// TwinCAT 3 PLC project SPS_Demonstrator
// ProgramVersion: 3.1.4026.19
// libraries:
//   Tc2_Standard, * (Beckhoff Automation GmbH)
//   Tc2_System, * (Beckhoff Automation GmbH)
//   Tc3_EventLogger, * (Beckhoff Automation GmbH)
//   Tc3_Module, * (Beckhoff Automation GmbH)
// project tree:
//   GVLs/ GVL.TcGVL, GVL_HRL.TcGVL, GVL_MBS.TcGVL, GVL_SST.TcGVL, GVL_VSG.TcGVL
//   / PlcTask.TcTTO
//   POUs/AtomicSkills/ Auto_ColorDetection.TcPOU, AxisControl_MultipleInputSensors.TcPOU, AxisControl_Encoder.TcPOU, CompressorControl.TcPOU, SecuringWorkpiece.TcPOU, StampingProcess.TcPOU, HardeningProcess.TcPOU, CuttingProcess.TcPOU
//   POUs/ControlOfOutputs/ HRL_ControlOfOutputs.TcPOU, MBS_ControlOfOutputs.TcPOU, SST_ControlOfOutputs.TcPOU, VSG_ControlOfOutputs.TcPOU
//   POUs/ HRL_SkillSet.TcPOU
//   POUs/MethodenBeispiele/ FB_MyOpcUaMethod.TcPOU, JobMethode_Schablone.TcPOU, HRL_NMethod_Auslagern.TcPOU, JobMethode.TcPOU
//   POUs/Moduls/HRL_Skills/ HRL_RGB_AS_VerticalMoveEncoder.TcPOU, HRL_RGB_AS_HorizontalMoveSensors.TcPOU, HRL_CB_AS_HorizontalMove.TcPOU, HRL_RGB_AS_HorizontalMoveEncoder.TcPOU, HRL_RGB_InitalStateDrive.TcPOU
//   POUs/Moduls/MBS_Skills/ MBS_MR01_AS_HardeningProcess.TcPOU, MBS_MR01_AS_SecuringProcess.TcPOU, MBS_VSG_AS_VerticalMove.TcPOU, MBS_MR01_AS_HorizontalMove.TcPOU, MBS_DmPD_AS_RotationMove.TcPOU, MBS_VSG_AS_HorizontalMove.TcPOU, MBS_CB_AS_HorizontalMove.TcPOU, MBS_DmPD_AS_HorizontalMove.TcPOU, MBS_MR02_AS_CuttingProcess.TcPOU
//   POUs/Moduls/SST_Skills/ SST_PD_AS_HorizontalMove.TcPOU, SST_CB_AS_HorizontalMove.TcPOU, SST_CS_AS_ColorDetection.TcPOU
//   POUs/Moduls/VSG_Skills/ VSG_AS_HorizontalMoveEncoder.TcPOU, VSG_AS_VerticalMoveEncoder.TcPOU, VSG_AS_RotationMoveEncoder.TcPOU, VSG_AS_CompressorControl.TcPOU
//   POUs/OperatingModes/ HRL_OperatingModes.TcPOU, MBS_OperatingModes.TcPOU, SST_OperatingModes.TcPOU, SVG_OperatingModes.TcPOU
// real-time tasks:
//   TASK PlcTask: cycle T#10ms, priority 20, ADS port 350
// I/O:
//   DEVICE Gerät 1 (EtherCAT), AmsNetId 5.152.132.139.2.1
//     Klemme 1 (EK1200) [EK1200-5000 EtherCAT Netzteil (2A E-Bus)]
//       Klemme 2 (EL1512) [EL1512 2K. +/- Zaehler 24V, 1kHz]
//       Klemme 3 (EL1512) [EL1512 2K. +/- Zaehler 24V, 1kHz]
//       Klemme 4 (EL1512) [EL1512 2K. +/- Zaehler 24V, 1kHz]
//       Klemme 5 (EL1512) [EL1512 2K. +/- Zaehler 24V, 1kHz]
//       Klemme 6 (EL1512) [EL1512 2K. +/- Zaehler 24V, 1kHz]
//       Klemme 7 (EL1409) [EL1409 16K. Dig. Eingang 24V, 3ms]
//       Klemme 8 (EL1409) [EL1409 16K. Dig. Eingang 24V, 3ms]
//       Klemme 9 (EL2409) [EL2409 16K. Dig. Ausgang 24V, 0.5A]
//       Klemme 10 (EL2409) [EL2409 16K. Dig. Ausgang 24V, 0.5A]
//       Klemme 11 (EL2008) [EL2008 8K. Dig. Ausgang 24V, 0.5A]
//       Klemme 12 (EL3072) [EL3072 2K. Ana. Eingang  +/-10V, +/-20mA]
//       Klemme 13 (EL9011) [EL9011 Endklemme]
// variable links:
//   SPS_Demonstrator/SPS_Demonstrator Instance <-> Device 1 (EtherCAT)/Term 1 (EK1200)/Term 10 (EL2409)
//     PlcTask Outputs/GVL_MBS.MBS_Kompressor <-> Channel 2/Output
//     PlcTask Outputs/GVL_MBS.MBS_Leuchte_Ofen <-> Channel 1/Output
//     PlcTask Outputs/GVL_MBS.MBS_MV_Ofentuer <-> Channel 5/Output
//     PlcTask Outputs/GVL_MBS.MBS_MV_Schieber <-> Channel 6/Output
//     PlcTask Outputs/GVL_MBS.MBS_MV_Vakuum <-> Channel 3/Output
//     PlcTask Outputs/GVL_MBS.MBS_MV_senken <-> Channel 4/Output
//     PlcTask Outputs/GVL_SST.SST_Kompressor <-> Channel 16/Output
//     PlcTask Outputs/GVL_SST.SST_MOT_Foerderband <-> Channel 15/Output
//     PlcTask Outputs/GVL_VSG.VSG_Kompressor <-> Channel 13/Output
//     PlcTask Outputs/GVL_VSG.VSG_MOT_drehen_CCW <-> Channel 12/Output
//     PlcTask Outputs/GVL_VSG.VSG_MOT_drehen_CW <-> Channel 11/Output
//     PlcTask Outputs/GVL_VSG.VSG_MOT_horizontal_rueckwaerts <-> Channel 9/Output
//     PlcTask Outputs/GVL_VSG.VSG_MOT_horizontal_vorwaerts <-> Channel 10/Output
//     PlcTask Outputs/GVL_VSG.VSG_MOT_vertikal_hoch <-> Channel 7/Output
//     PlcTask Outputs/GVL_VSG.VSG_MOT_vertikal_runter <-> Channel 8/Output
//     PlcTask Outputs/GVL_VSG.VSG_MV_Vakuum <-> Channel 14/Output
//   SPS_Demonstrator/SPS_Demonstrator Instance <-> Device 1 (EtherCAT)/Term 1 (EK1200)/Term 11 (EL2008)
//     PlcTask Outputs/GVL_SST.SST_MV_blau <-> Channel 3/Output
//     PlcTask Outputs/GVL_SST.SST_MV_rot <-> Channel 2/Output
//     PlcTask Outputs/GVL_SST.SST_MV_weiss <-> Channel 1/Output
//   SPS_Demonstrator/SPS_Demonstrator Instance <-> Device 1 (EtherCAT)/Term 1 (EK1200)/Term 12 (EL3072)
//     PlcTask Inputs/GVL_SST.SST_Farbsensor <-> AI Standard Channel 1/Value
//   SPS_Demonstrator/SPS_Demonstrator Instance <-> Device 1 (EtherCAT)/Term 1 (EK1200)/Term 2 (EL1512)
//     PlcTask Inputs/GVL_HRL.HRL_Enc_horizontal_I1 <-> CNT Inputs Channel 1/Counter value
//     PlcTask Inputs/GVL_HRL.HRL_Enc_horizontal_I2 <-> CNT Inputs Channel 2/Counter value
//     PlcTask Outputs/GVL_HRL.HRL_K1_1_Zaehler_Zuruecksetzen <-> CNT Outputs Channel 1/Control/Set counter
//   SPS_Demonstrator/SPS_Demonstrator Instance <-> Device 1 (EtherCAT)/Term 1 (EK1200)/Term 3 (EL1512)
//     PlcTask Inputs/GVL_HRL.HRL_Enc_vertikal_I1 <-> CNT Inputs Channel 1/Counter value
//     PlcTask Inputs/GVL_HRL.HRL_Enc_vertikal_I2 <-> CNT Inputs Channel 2/Counter value
//     PlcTask Outputs/GVL_HRL.HRL_K1_2_Zaehler_Zuruecksetzen <-> CNT Outputs Channel 1/Control/Set counter
//   SPS_Demonstrator/SPS_Demonstrator Instance <-> Device 1 (EtherCAT)/Term 1 (EK1200)/Term 4 (EL1512)
//     PlcTask Inputs/GVL_VSG.VSG_Enc_vertikal_I1 <-> CNT Inputs Channel 1/Counter value
//     PlcTask Inputs/GVL_VSG.VSG_Enc_vertikal_I2 <-> CNT Inputs Channel 2/Counter value
//     PlcTask Outputs/GVL_VSG.VSG_K1_3_Zaehler_Zuruecksetzen <-> CNT Outputs Channel 1/Control/Set counter
//   SPS_Demonstrator/SPS_Demonstrator Instance <-> Device 1 (EtherCAT)/Term 1 (EK1200)/Term 5 (EL1512)
//     PlcTask Inputs/GVL_VSG.VSG_Enc_horizontal_I1 <-> CNT Inputs Channel 1/Counter value
//     PlcTask Inputs/GVL_VSG.VSG_Enc_horizontal_I2 <-> CNT Inputs Channel 2/Counter value
//     PlcTask Outputs/GVL_VSG.VSG_K1_4_Zaehler_Zuruecksetzen <-> CNT Outputs Channel 1/Set counter
//   SPS_Demonstrator/SPS_Demonstrator Instance <-> Device 1 (EtherCAT)/Term 1 (EK1200)/Term 6 (EL1512)
//     PlcTask Inputs/GVL_VSG.VSG_Enc_drehen_I1 <-> CNT Inputs Channel 1/Counter value
//     PlcTask Inputs/GVL_VSG.VSG_Enc_drehen_I2 <-> CNT Inputs Channel 2/Counter value
//     PlcTask Outputs/GVL_VSG.VSG_K1_5_Zaehler_Zuruecksetzen <-> CNT Outputs Channel 1/Control/Set counter
//   SPS_Demonstrator/SPS_Demonstrator Instance <-> Device 1 (EtherCAT)/Term 1 (EK1200)/Term 7 (EL1409)
//     PlcTask Inputs/GVL_HRL.HRL_LS_aussen <-> DIP Inputs/Input Channel 3
//     PlcTask Inputs/GVL_HRL.HRL_LS_innen <-> DIP Inputs/Input Channel 2
//     PlcTask Inputs/GVL_HRL.HRL_Ref_Taster_Ausleger_hinten <-> DIP Inputs/Input Channel 8
//     PlcTask Inputs/GVL_HRL.HRL_Ref_Taster_Ausleger_vorne <-> DIP Inputs/Input Channel 7
//     PlcTask Inputs/GVL_HRL.HRL_Ref_Taster_horizontal <-> DIP Inputs/Input Channel 1
//     PlcTask Inputs/GVL_HRL.HRL_Ref_Taster_vertikal <-> DIP Inputs/Input Channel 4
//     PlcTask Inputs/GVL_HRL.HRL_Spursensor_1_unten <-> DIP Inputs/Input Channel 5
//     PlcTask Inputs/GVL_HRL.HRL_Spursensor_2_oben <-> DIP Inputs/Input Channel 6
//     PlcTask Inputs/GVL_MBS.MBS_LS_Ende_Foerderband <-> DIP Inputs/Input Channel 11
//     PlcTask Inputs/GVL_MBS.MBS_Ref_Taster_DK_Pos_Foerderband <-> DIP Inputs/Input Channel 10
//     PlcTask Inputs/GVL_MBS.MBS_Ref_Taster_DK_Pos_Saege <-> DIP Inputs/Input Channel 12
//     PlcTask Inputs/GVL_MBS.MBS_Ref_Taster_DK_Pos_Sauger <-> DIP Inputs/Input Channel 9
//     PlcTask Inputs/GVL_MBS.MBS_Ref_Taster_Ofenschieber_aussen <-> DIP Inputs/Input Channel 15
//     PlcTask Inputs/GVL_MBS.MBS_Ref_Taster_Ofenschieber_innen <-> DIP Inputs/Input Channel 14
//     PlcTask Inputs/GVL_MBS.MBS_Ref_Taster_Sauger_Pos_DK <-> DIP Inputs/Input Channel 13
//     PlcTask Inputs/GVL_MBS.MBS_Ref_Taster_Sauger_Pos_Ofen <-> DIP Inputs/Input Channel 16
//   SPS_Demonstrator/SPS_Demonstrator Instance <-> Device 1 (EtherCAT)/Term 1 (EK1200)/Term 8 (EL1409)
//     PlcTask Inputs/GVL.diNotAus_Kanal_A <-> DIP Inputs/Input Channel 11
//     PlcTask Inputs/GVL.diNotAus_Kanal_B <-> DIP Inputs/Input Channel 12
//     PlcTask Inputs/GVL_MBS.MBS_LS_Ofen <-> DIP Inputs/Input Channel 1
//     PlcTask Inputs/GVL_SST.SST_Impulstaster <-> DIP Inputs/Input Channel 5
//     PlcTask Inputs/GVL_SST.SST_LS_Eingang <-> DIP Inputs/Input Channel 6
//     PlcTask Inputs/GVL_SST.SST_LS_blau <-> DIP Inputs/Input Channel 10
//     PlcTask Inputs/GVL_SST.SST_LS_nach_Farbsensor <-> DIP Inputs/Input Channel 7
//     PlcTask Inputs/GVL_SST.SST_LS_rot <-> DIP Inputs/Input Channel 9
//     PlcTask Inputs/GVL_SST.SST_LS_weiss <-> DIP Inputs/Input Channel 8
//     PlcTask Inputs/GVL_VSG.VSG_Ref_Schalter_drehen <-> DIP Inputs/Input Channel 4
//     PlcTask Inputs/GVL_VSG.VSG_Ref_Schalter_horizontal <-> DIP Inputs/Input Channel 3
//     PlcTask Inputs/GVL_VSG.VSG_Ref_Schalter_vertikal <-> DIP Inputs/Input Channel 2
//   SPS_Demonstrator/SPS_Demonstrator Instance <-> Device 1 (EtherCAT)/Term 1 (EK1200)/Term 9 (EL2409)
//     PlcTask Outputs/GVL_HRL.HRL_MOT_Ausleger_rueckwaerts <-> Channel 8/Output
//     PlcTask Outputs/GVL_HRL.HRL_MOT_Ausleger_vorwaerts <-> Channel 7/Output
//     PlcTask Outputs/GVL_HRL.HRL_MOT_Foerderband_rueckwaerts <-> Channel 2/Output
//     PlcTask Outputs/GVL_HRL.HRL_MOT_Foerderband_vorwaerts <-> Channel 1/Output
//     PlcTask Outputs/GVL_HRL.HRL_MOT_horizontal_zum_Foerderband <-> Channel 4/Output
//     PlcTask Outputs/GVL_HRL.HRL_MOT_horizontal_zum_Regal <-> Channel 3/Output
//     PlcTask Outputs/GVL_HRL.HRL_MOT_vertikal_hoch <-> Channel 6/Output
//     PlcTask Outputs/GVL_HRL.HRL_MOT_vertikal_runter <-> Channel 5/Output
//     PlcTask Outputs/GVL_MBS.MBS_MOT_DK_CCW <-> Channel 10/Output
//     PlcTask Outputs/GVL_MBS.MBS_MOT_DK_CW <-> Channel 9/Output
//     PlcTask Outputs/GVL_MBS.MBS_MOT_Foerderband_vorwaerts <-> Channel 11/Output
//     PlcTask Outputs/GVL_MBS.MBS_MOT_Ofenschieber_ausfahren <-> Channel 14/Output
//     PlcTask Outputs/GVL_MBS.MBS_MOT_Ofenschieber_einfahren <-> Channel 13/Output
//     PlcTask Outputs/GVL_MBS.MBS_MOT_Saege <-> Channel 12/Output
//     PlcTask Outputs/GVL_MBS.MBS_MOT_Sauger_zum_DK <-> Channel 16/Output
//     PlcTask Outputs/GVL_MBS.MBS_MOT_Sauger_zum_Ofen <-> Channel 15/Output

CONFIGURATION SPS_Demonstrator
    RESOURCE PLC ON TwinCAT3
        TASK PlcTask(INTERVAL := T#10ms, PRIORITY := 20);
        PROGRAM InitalizingOM WITH PlcTask : InitalizingOM;
        PROGRAM HRL_SkillSet WITH PlcTask : HRL_SkillSet;
    END_RESOURCE
END_CONFIGURATION

// ---- GVLs/GVL.TcGVL
{attribute 'qualified_only'}
VAR_GLOBAL
	// xDI%139.2_S1_2
	diNotAus_Kanal_A AT %I*: BOOL;
	// xDI%139.3_S1_2
	diNotAus_Kanal_B AT %I*: BOOL;
END_VAR

// ---- GVLs/GVL_HRL.TcGVL
{attribute 'qualified_only'}
VAR_GLOBAL
	// udiDI%41.0_A2_5
	HRL_Enc_horizontal_I1 AT %I*: UDINT;
	// udiDI%47.0_A2_5
	HRL_Enc_horizontal_I2 AT %I*: UDINT;
	// udiDI%53.0_A2_5
	HRL_Enc_vertikal_I1 AT %I*: UDINT;
	// udiDI%59.0_A2_5
	HRL_Enc_vertikal_I2 AT %I*: UDINT;
	// xDI%136.0_A2_2
	HRL_Ref_Taster_horizontal AT %I*: BOOL;
	// xDI%136.1_A2_1
	HRL_LS_innen AT %I*: BOOL;
	// xDI%136.2_A2_1
	HRL_LS_aussen AT %I*: BOOL;
	// xDI%136.3_A2_2
	HRL_Ref_Taster_vertikal AT %I*: BOOL;
	// xDI%136.4_A2_3
	HRL_Spursensor_1_unten AT %I*: BOOL;
	// xDI%136.5_A2_3
	HRL_Spursensor_2_oben AT %I*: BOOL;
	// xDI%136.6_A2_2
	HRL_Ref_Taster_Ausleger_vorne AT %I*: BOOL;
	// xDI%136.7_A2_2
	HRL_Ref_Taster_Ausleger_hinten AT %I*: BOOL;
	// xDO%111.0_A2_2	
	HRL_MOT_Foerderband_vorwaerts AT %Q*: BOOL;
	// xDO%111.1_A2_2
	HRL_MOT_Foerderband_rueckwaerts AT %Q*: BOOL;
	// xDO%111.2_A2_4
	HRL_MOT_horizontal_zum_Regal AT %Q*: BOOL;
	// xDO%111.3_A2_4
	HRL_MOT_horizontal_zum_Foerderband AT %Q*: BOOL;
	// xDO%111.4_A2_4
	HRL_MOT_vertikal_runter AT %Q*: BOOL;
	// xDO%111.5_A2_4
	HRL_MOT_vertikal_hoch AT %Q*: BOOL;
	// xDO%111.6_A2_4
	HRL_MOT_Ausleger_vorwaerts AT %Q*: BOOL;
	// xDO%111.7_A2_4
	HRL_MOT_Ausleger_rueckwaerts AT %Q*: BOOL;
	HRL_K1_1_Zaehler_Zuruecksetzen AT %Q*: BOOL;
	HRL_K1_2_Zaehler_Zuruecksetzen AT %Q*: BOOL;
END_VAR

// ---- GVLs/GVL_MBS.TcGVL
{attribute 'qualified_only'}
VAR_GLOBAL
	// xDI%137.0_A3_2
	MBS_Ref_Taster_DK_Pos_Sauger AT %I*: BOOL;
	// xDI%137.1_A3_2
	MBS_Ref_Taster_DK_Pos_Foerderband AT %I*: BOOL;
	// xDI%137.2_A3_1
	MBS_LS_Ende_Foerderband AT %I*: BOOL;
	// xDI%137.3_A3_2
	MBS_Ref_Taster_DK_Pos_Saege AT %I*: BOOL;
	// xDI%137.4_A3_2
	MBS_Ref_Taster_Sauger_Pos_DK AT %I*: BOOL;
	// xDI%137.5_A3_2
	MBS_Ref_Taster_Ofenschieber_innen AT %I*: BOOL;
	// xDI%137.6_A3_2
	MBS_Ref_Taster_Ofenschieber_aussen AT %I*: BOOL;
	// xDI%137.7_A3_2
	MBS_Ref_Taster_Sauger_Pos_Ofen AT %I*: BOOL;
	// xDI%138.0_A3_1
	MBS_LS_Ofen AT %I*: BOOL;
	// xDO%112.0_A3_4
	MBS_MOT_DK_CW AT %Q*: BOOL;
	// xDO%112.1_A3_4
	MBS_MOT_DK_CCW AT %Q*: BOOL;
	// xDO%112.2_A3_2
	MBS_MOT_Foerderband_vorwaerts AT %Q*: BOOL;
	// xDO%112.3_A3_6
	MBS_MOT_Saege AT %Q*: BOOL;
	// xDO%112.4_A3_3
	MBS_MOT_Ofenschieber_einfahren AT %Q*: BOOL;
	// xDO%112.5_A3_3
	MBS_MOT_Ofenschieber_ausfahren AT %Q*: BOOL;
	// xDO%112.6_A3_5
	MBS_MOT_Sauger_zum_Ofen AT %Q*: BOOL;
	// xDO%112.7_A3_5
	MBS_MOT_Sauger_zum_DK AT %Q*: BOOL;
	// xDO%113.0_A3_7
	MBS_Leuchte_Ofen AT %Q*: BOOL;
	// xDO%113.1_A3_8
	MBS_Kompressor AT %Q*: BOOL;
	// xDO%113.2_A3_5
	MBS_MV_Vakuum AT %Q*: BOOL;
	// xDO%113.3_A3_5
	MBS_MV_senken AT %Q*: BOOL;
	// xDO%113.4_A3_5
	MBS_MV_Ofentuer AT %Q*: BOOL;
	// xDO%113.5_A3_5
	MBS_MV_Schieber AT %Q*: BOOL;
END_VAR

// ---- GVLs/GVL_SST.TcGVL
{attribute 'qualified_only'}
VAR_GLOBAL
	// xDO%115.0_A5_5
	SST_MV_weiss AT %Q*: BOOL;
	// xDO%115.1_A5_5
	SST_MV_rot AT %Q*: BOOL;
	// xDO%115.2_A5_5
	SST_MV_blau AT %Q*: BOOL;
	// iAI%130.0_A5_4
	SST_Farbsensor AT %I*: INT;
	// xDI%138.4_A5_1
	SST_Impulstaster AT %I*: BOOL;
	// xDI%138.5_A5_1
	SST_LS_Eingang AT %I*: BOOL;
	// xDI%138.6_A5_1
	SST_LS_nach_Farbsensor AT %I*: BOOL;
	// xDI%138.7_A5_1
	SST_LS_weiss AT %I*: BOOL;
	// xDI%139.0_A5_1
	SST_LS_rot AT %I*: BOOL;
	// xDI%139.1_A5_1
	SST_LS_blau AT %I*: BOOL;
	// xDO%114.6_A5_2
	SST_MOT_Foerderband AT %Q*: BOOL;
	// xDO%114.7_A5_8
	SST_Kompressor AT %Q*: BOOL;
END_VAR

// ---- GVLs/GVL_VSG.TcGVL
{attribute 'qualified_only'}
VAR_GLOBAL
	// udiDI%65.0_A4_5
	VSG_Enc_vertikal_I1 AT %I*: UDINT;
	// udiDI%71.0_A4_5
	VSG_Enc_vertikal_I2 AT %I*: UDINT;
	// udiDI%77.0_A4_5
	VSG_Enc_horizontal_I1 AT %I*: UDINT;
	// udiDI%83.0_A4_5
	VSG_Enc_horizontal_I2 AT %I*: UDINT;
	// udiDI%89.0_A4_5
	VSG_Enc_drehen_I1 AT %I*: UDINT;
	// udiDI%95.0_A4_5
	VSG_Enc_drehen_I2 AT %I*: UDINT;
	// xDI%138.1_A4_2
	VSG_Ref_Schalter_vertikal AT %I*: BOOL;
	// xDI%138.2_A4_2
	VSG_Ref_Schalter_horizontal AT %I*: BOOL;
	// xDI%138.3_A4_2
	VSG_Ref_Schalter_drehen AT %I*: BOOL;
	// xDO%113.6_A4_4
	VSG_MOT_vertikal_hoch AT %Q*: BOOL;
	// xDO%113.7_A4_4
	VSG_MOT_vertikal_runter AT %Q*: BOOL;
	// xDO%114.0_A4_4
	VSG_MOT_horizontal_rueckwaerts AT %Q*: BOOL;
	// xDO%114.1_A4_4
	VSG_MOT_horizontal_vorwaerts AT %Q*: BOOL;
	// xDO%114.2_A4_4
	VSG_MOT_drehen_CW AT %Q*: BOOL;
	// xDO%114.3_A4_4
	VSG_MOT_drehen_CCW AT %Q*: BOOL;
	// xDO%114.4_A4_8
	VSG_Kompressor AT %Q*: BOOL;
	// xDO%114.5_A4_5
	VSG_MV_Vakuum AT %Q*: BOOL;
	VSG_K1_4_Zaehler_Zuruecksetzen AT %Q*: BOOL;
	VSG_K1_5_Zaehler_Zuruecksetzen AT %Q*: BOOL;
	VSG_K1_3_Zaehler_Zuruecksetzen AT %Q*: BOOL;
END_VAR

// ---- POUs/HRL_SkillSet.TcPOU
PROGRAM HRL_SkillSet
VAR
//Hochregallager Skillset	
	
	//HRL Conveyorbelt Skills
	{attribute 'OPC.UA.DA':= '1'}
	HRL_Skill_CB_MoveForwards: HRL_CB_AS_HorizontalMove; //Movement to Store-Out some goods on the Conveyorbelt
	{attribute 'OPC.UA.DA':= '1'}
	HRL_Skill_CB_MoveBackwards : HRL_CB_AS_HorizontalMove; //Movement to Store-In some goods on the Conveyorbelt
	
	//HRL RGB Skills
	{attribute 'OPC.UA.DA':= '1'}
	HRL_Skill_RGB_MoveBackwards : HRL_RGB_AS_HorizontalMoveSensors;	
	{attribute 'OPC.UA.DA':= '1'}
	HRL_Skill_RGB_MoveForwards : HRL_RGB_AS_HorizontalMoveSensors;	
	{attribute 'OPC.UA.DA':= '1'}
	HRL_Skill_RGB_MoveVerticalForwards : HRL_RGB_AS_VerticalMoveEncoder;	
	{attribute 'OPC.UA.DA':= '1'}
	HRL_Skill_RGB_MoveVerticalBackwards : HRL_RGB_AS_VerticalMoveEncoder;
	{attribute 'OPC.UA.DA':= '1'}
	HRL_Skill_RGB_MoveHorizontalForwards : HRL_RGB_AS_HorizontalMoveEncoder;	
	{attribute 'OPC.UA.DA':= '1'}
	HRL_Skill_RGB_MoveHorizontalBackwards : HRL_RGB_AS_HorizontalMoveEncoder;
	
	HRL_ControlOfOutputs : HRL_COntrolOfOutputs;
	HRL_OperatingModes : HRL_OperatingModes;
//TestMethode NMethode für Auslagern //
	{attribute 'OPC.UA.DA':= '1'}
	HRL_NMethod_Auslagern :HRL_NMethod_Auslagern;

//Variablensetzung: Sollte später über SkillOA eingesetzt werden ODER Hard in SPS codiert (Diskussionspunkt)
	TIME_TSR : TIME := T#150MS;
	ResetButton: BOOL;
	StartButton: BOOL;
	ConfirmationButton: BOOL;
END_VAR

VAR_OUTPUT
	HRL_CB_forwards : BOOL; //GVL_HRL.HRL_MOT_Foerderband_vorwaerts
	HRL_CB_backwards : BOOL; //GVL_HRL.HRL_MOT_Foerderband_rueckwaerts
	HRL_RGB_Forwards01 : BOOL; //GVL_HRL.HRL_MOT_Ausleger_vorwaerts
	HRL_RGB_Forwards02 : BOOL; //GVL_HRL.HRL_MOT_Ausleger_rueckwaerts
	HRL_RGB_Backwards01 : BOOL; //GVL_HRL.HRL_MOT_Ausleger_rueckwaerts
	HRL_RGB_Backwards02 : BOOL; //GVL_HRL.HRL_MOT_Ausleger_vorwaerts
	HRL_RGB_VertikalDown01 : BOOL; //GVL_HRL.HRL_MOT_vertikal_runter
	HRL_RGB_VertikalDown02 : BOOL; //GVL_HRL.HRL_MOT_vertikal_hoch
	HRL_RGB_VertikalUp01 : BOOL; //GVL_HRL.HRL_MOT_vertikal_hoch
	HRL_RGB_VertikalUp02 : BOOL; //GVL_HRL.HRL_MOT_vertikal_runter
	HRL_RGB_HorizontalForwards01 : BOOL; //GVL_HRL.HRL_MOT_horizontal_zum_Regal
	HRL_RGB_HorizontalForwards02 : BOOL; //GVL_HRL.HRL_MOT_horizontal_zum_Foerderband
	HRL_RGB_HorizontalBackwards01 : BOOL; //GVL_HRL.HRL_MOT_horizontal_zum_Foerderband
	HRL_RGB_HorizontalBackwards02 : BOOL; //GVL_HRL.HRL_MOT_horizontal_zum_Regal
END_VAR

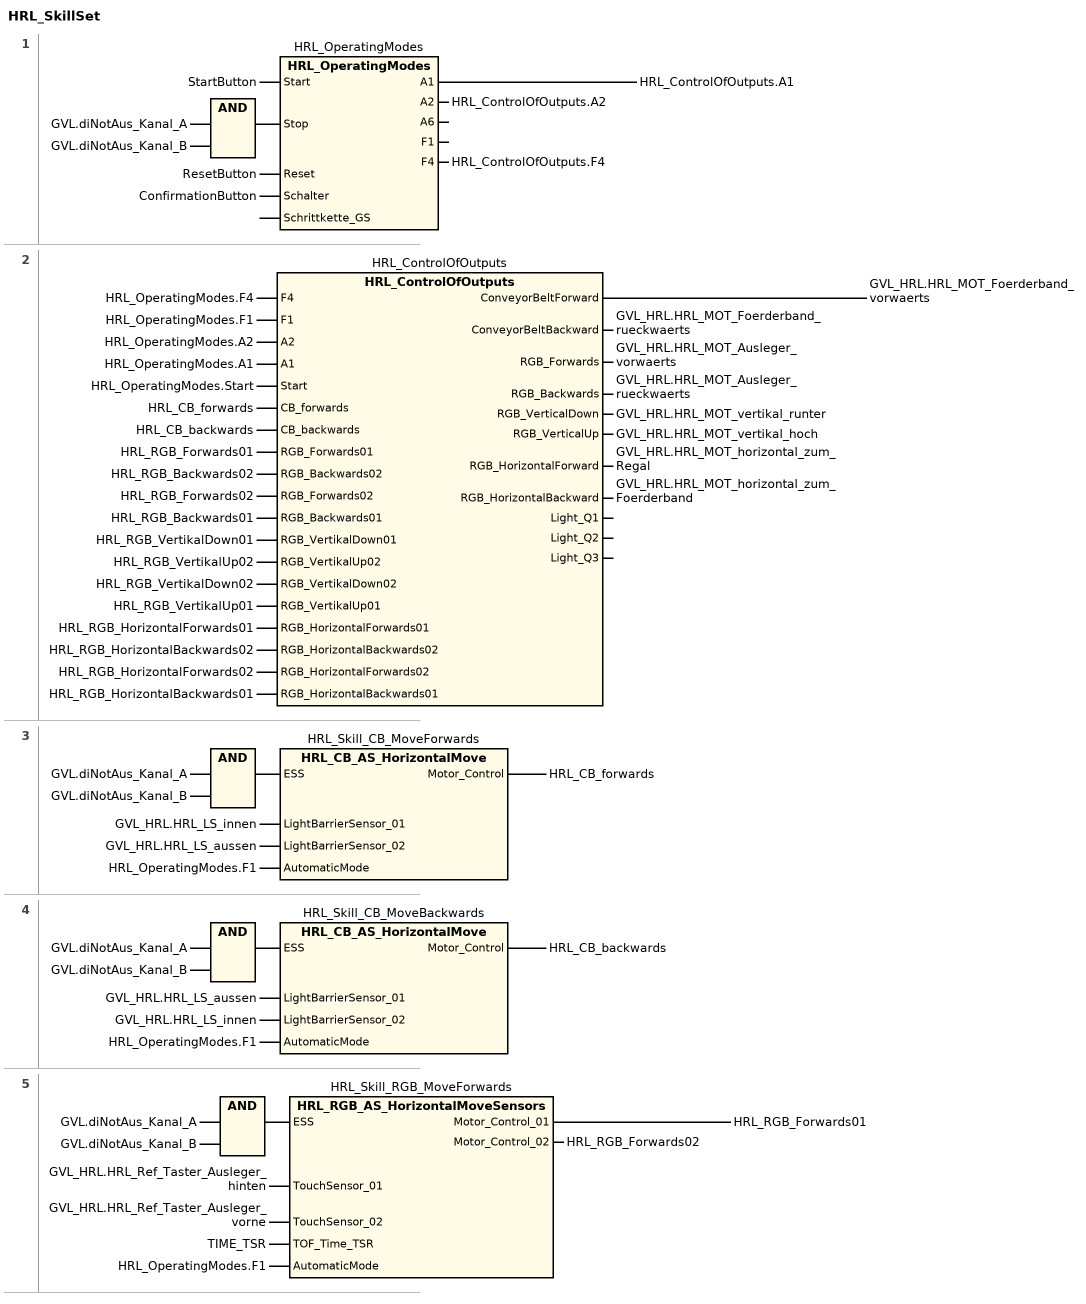
// NETWORK 1
HRL_OperatingModes(
    Start := StartButton,
    Stop := GVL.diNotAus_Kanal_A AND GVL.diNotAus_Kanal_B,
    Reset := ResetButton,
    Schalter := ConfirmationButton,
    A2 => HRL_ControlOfOutputs.A2,
    F4 => HRL_ControlOfOutputs.F4);
HRL_ControlOfOutputs.A1 := HRL_OperatingModes.A1;

// NETWORK 2
HRL_ControlOfOutputs(
    F4 := HRL_OperatingModes.F4,
    F1 := HRL_OperatingModes.F1,
    A2 := HRL_OperatingModes.A2,
    A1 := HRL_OperatingModes.A1,
    Start := HRL_OperatingModes.Start,
    CB_forwards := HRL_CB_forwards,
    CB_backwards := HRL_CB_backwards,
    RGB_Forwards01 := HRL_RGB_Forwards01,
    RGB_Backwards02 := HRL_RGB_Backwards02,
    RGB_Forwards02 := HRL_RGB_Forwards02,
    RGB_Backwards01 := HRL_RGB_Backwards01,
    RGB_VertikalDown01 := HRL_RGB_VertikalDown01,
    RGB_VertikalUp02 := HRL_RGB_VertikalUp02,
    RGB_VertikalDown02 := HRL_RGB_VertikalDown02,
    RGB_VertikalUp01 := HRL_RGB_VertikalUp01,
    RGB_HorizontalForwards01 := HRL_RGB_HorizontalForwards01,
    RGB_HorizontalBackwards02 := HRL_RGB_HorizontalBackwards02,
    RGB_HorizontalForwards02 := HRL_RGB_HorizontalForwards02,
    RGB_HorizontalBackwards01 := HRL_RGB_HorizontalBackwards01,
    ConveyorBeltBackward => GVL_HRL.HRL_MOT_Foerderband_rueckwaerts,
    RGB_Forwards => GVL_HRL.HRL_MOT_Ausleger_vorwaerts,
    RGB_Backwards => GVL_HRL.HRL_MOT_Ausleger_rueckwaerts,
    RGB_VerticalDown => GVL_HRL.HRL_MOT_vertikal_runter,
    RGB_VerticalUp => GVL_HRL.HRL_MOT_vertikal_hoch,
    RGB_HorizontalForward => GVL_HRL.HRL_MOT_horizontal_zum_Regal,
    RGB_HorizontalBackward => GVL_HRL.HRL_MOT_horizontal_zum_Foerderband);
GVL_HRL.HRL_MOT_Foerderband_vorwaerts := HRL_ControlOfOutputs.ConveyorBeltForward;

// NETWORK 3
HRL_Skill_CB_MoveForwards(
    ESS := GVL.diNotAus_Kanal_A AND GVL.diNotAus_Kanal_B,
    LightBarrierSensor_01 := GVL_HRL.HRL_LS_innen,
    LightBarrierSensor_02 := GVL_HRL.HRL_LS_aussen,
    AutomaticMode := HRL_OperatingModes.F1); // HRL_CB_AS_HorizontalMove
HRL_CB_forwards := HRL_Skill_CB_MoveForwards.Motor_Control;

// NETWORK 4
HRL_Skill_CB_MoveBackwards(
    ESS := GVL.diNotAus_Kanal_A AND GVL.diNotAus_Kanal_B,
    LightBarrierSensor_01 := GVL_HRL.HRL_LS_aussen,
    LightBarrierSensor_02 := GVL_HRL.HRL_LS_innen,
    AutomaticMode := HRL_OperatingModes.F1); // HRL_CB_AS_HorizontalMove
HRL_CB_backwards := HRL_Skill_CB_MoveBackwards.Motor_Control;

// NETWORK 5
HRL_Skill_RGB_MoveForwards(
    ESS := GVL.diNotAus_Kanal_A AND GVL.diNotAus_Kanal_B,
    TouchSensor_01 := GVL_HRL.HRL_Ref_Taster_Ausleger_hinten,
    TouchSensor_02 := GVL_HRL.HRL_Ref_Taster_Ausleger_vorne,
    TOF_Time_TSR := TIME_TSR,
    AutomaticMode := HRL_OperatingModes.F1,
    Motor_Control_02 => HRL_RGB_Forwards02); // HRL_RGB_AS_HorizontalMoveSensors
HRL_RGB_Forwards01 := HRL_Skill_RGB_MoveForwards.Motor_Control_01;

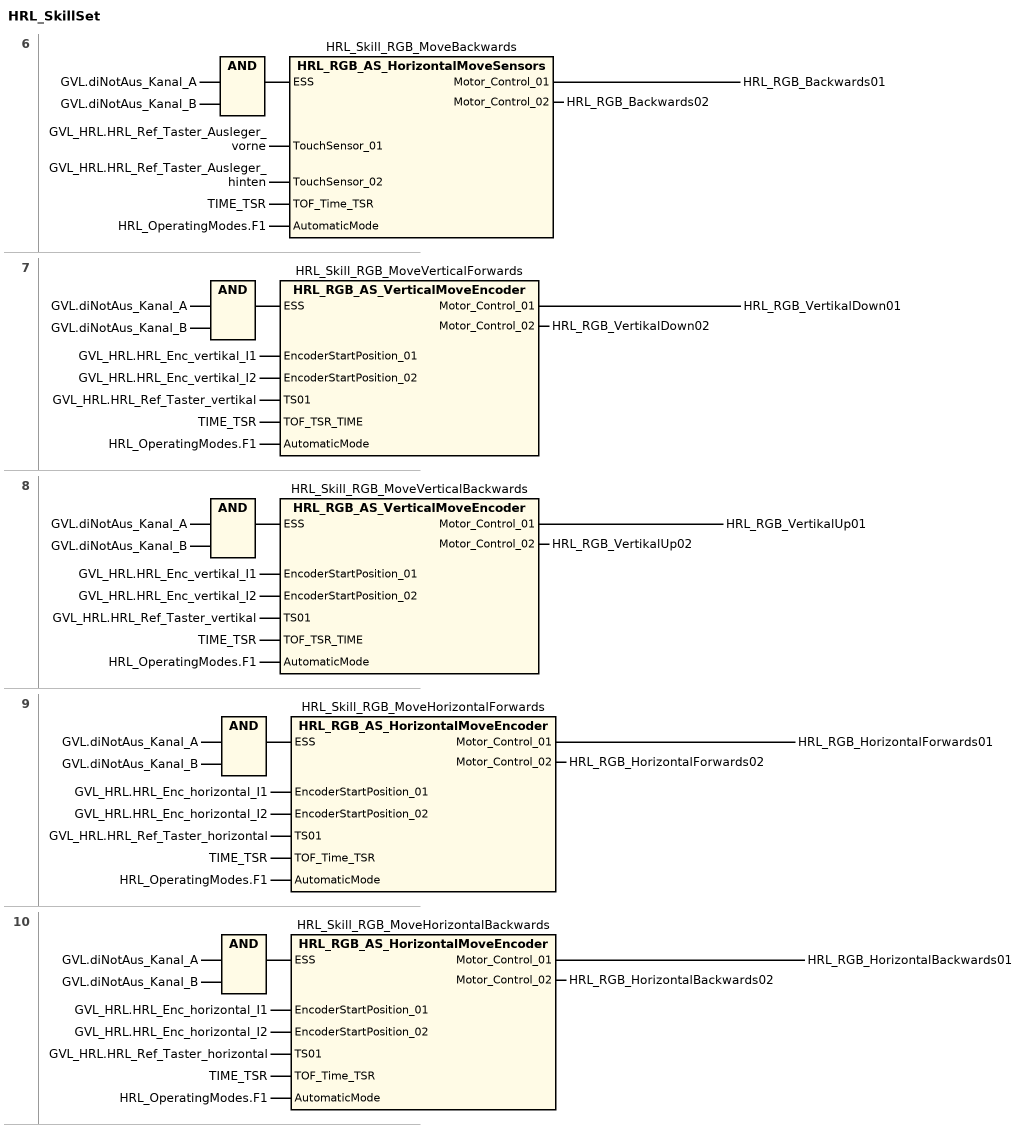
// NETWORK 6
HRL_Skill_RGB_MoveBackwards(
    ESS := GVL.diNotAus_Kanal_A AND GVL.diNotAus_Kanal_B,
    TouchSensor_01 := GVL_HRL.HRL_Ref_Taster_Ausleger_vorne,
    TouchSensor_02 := GVL_HRL.HRL_Ref_Taster_Ausleger_hinten,
    TOF_Time_TSR := TIME_TSR,
    AutomaticMode := HRL_OperatingModes.F1,
    Motor_Control_02 => HRL_RGB_Backwards02); // HRL_RGB_AS_HorizontalMoveSensors
HRL_RGB_Backwards01 := HRL_Skill_RGB_MoveBackwards.Motor_Control_01;

// NETWORK 7
HRL_Skill_RGB_MoveVerticalForwards(
    ESS := GVL.diNotAus_Kanal_A AND GVL.diNotAus_Kanal_B,
    EncoderStartPosition_01 := GVL_HRL.HRL_Enc_vertikal_I1,
    EncoderStartPosition_02 := GVL_HRL.HRL_Enc_vertikal_I2,
    TS01 := GVL_HRL.HRL_Ref_Taster_vertikal,
    TOF_TSR_TIME := TIME_TSR,
    AutomaticMode := HRL_OperatingModes.F1,
    Motor_Control_02 => HRL_RGB_VertikalDown02); // HRL_RGB_AS_VerticalMoveEncoder
HRL_RGB_VertikalDown01 := HRL_Skill_RGB_MoveVerticalForwards.Motor_Control_01;

// NETWORK 8
HRL_Skill_RGB_MoveVerticalBackwards(
    ESS := GVL.diNotAus_Kanal_A AND GVL.diNotAus_Kanal_B,
    EncoderStartPosition_01 := GVL_HRL.HRL_Enc_vertikal_I1,
    EncoderStartPosition_02 := GVL_HRL.HRL_Enc_vertikal_I2,
    TS01 := GVL_HRL.HRL_Ref_Taster_vertikal,
    TOF_TSR_TIME := TIME_TSR,
    AutomaticMode := HRL_OperatingModes.F1,
    Motor_Control_02 => HRL_RGB_VertikalUp02); // HRL_RGB_AS_VerticalMoveEncoder
HRL_RGB_VertikalUp01 := HRL_Skill_RGB_MoveVerticalBackwards.Motor_Control_01;

// NETWORK 9
HRL_Skill_RGB_MoveHorizontalForwards(
    ESS := GVL.diNotAus_Kanal_A AND GVL.diNotAus_Kanal_B,
    EncoderStartPosition_01 := GVL_HRL.HRL_Enc_horizontal_I1,
    EncoderStartPosition_02 := GVL_HRL.HRL_Enc_horizontal_I2,
    TS01 := GVL_HRL.HRL_Ref_Taster_horizontal,
    TOF_Time_TSR := TIME_TSR,
    AutomaticMode := HRL_OperatingModes.F1,
    Motor_Control_02 => HRL_RGB_HorizontalForwards02); // HRL_RGB_AS_HorizontalMoveEncoder
HRL_RGB_HorizontalForwards01 := HRL_Skill_RGB_MoveHorizontalForwards.Motor_Control_01;

// NETWORK 10
HRL_Skill_RGB_MoveHorizontalBackwards(
    ESS := GVL.diNotAus_Kanal_A AND GVL.diNotAus_Kanal_B,
    EncoderStartPosition_01 := GVL_HRL.HRL_Enc_horizontal_I1,
    EncoderStartPosition_02 := GVL_HRL.HRL_Enc_horizontal_I2,
    TS01 := GVL_HRL.HRL_Ref_Taster_horizontal,
    TOF_Time_TSR := TIME_TSR,
    AutomaticMode := HRL_OperatingModes.F1,
    Motor_Control_02 => HRL_RGB_HorizontalBackwards02); // HRL_RGB_AS_HorizontalMoveEncoder
HRL_RGB_HorizontalBackwards01 := HRL_Skill_RGB_MoveHorizontalBackwards.Motor_Control_01;

END_PROGRAM

// ---- POUs/Moduls/HRL_Skills/HRL_CB_AS_HorizontalMove.TcPOU
{attribute 'OPC.UA.DA.JobMethod' := 'JobMethode_HorizontalMove'}
FUNCTION_BLOCK HRL_CB_AS_HorizontalMove
VAR
	AlwaysTrue : BOOL := TRUE;
	// Used for debugging purposes to display InputArguments of method call
	MethodCall_HorizontalMove : BOOL := FALSE; // used to store InputArg "MethodCall" from Start() method
	ResetMethodCall	: BOOL := FALSE;
	Direction : BOOL := FALSE; // defines movement direction
	callCounterStart : ULINT; // counts how many times the Start() method has been called
	callCounterCheckState : ULINT; // counts how many times the CheckState() method has been called
	callCounterAbort : ULINT; // counts how many times the Abort() method has been called
	
	// Variables to determine if a job has been started (Start() method has been called) or finished
	jobRunning : BOOL;
	jobFinished : BOOL;

	// State machine variable
	state : UDINT;
	
	// FB Intatziation Variable
	HRL_CB_HorizontalMove : AxisControl_MultipleInputSensors;
END_VAR
	
VAR_INPUT
	ESS: BOOL;
	LightBarrierSensor_01 : BOOL;
	LightBarrierSensor_02 : BOOL;
	AutomaticMode: BOOL;
END_VAR

VAR_OUTPUT
	Motor_Control : BOOL;
END_VAR

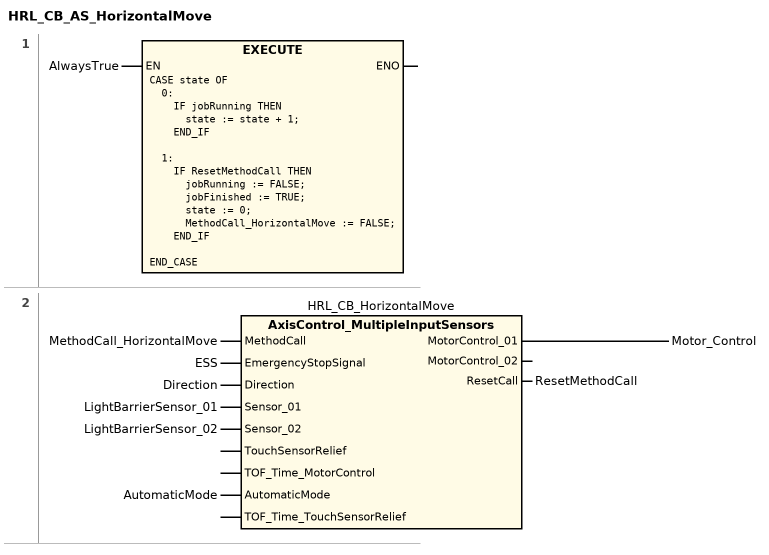
// NETWORK 1
IF AlwaysTrue THEN
    CASE state OF
    	0:
    		IF jobRunning THEN
    			state := state + 1;
    		END_IF
    		
    	1:
    		IF ResetMethodCall THEN
    			jobRunning := FALSE;
    			jobFinished := TRUE;
    			state := 0;
    			MethodCall_HorizontalMove := FALSE;
    		END_IF
    		
    END_CASE
END_IF

// NETWORK 2
HRL_CB_HorizontalMove(
    MethodCall := MethodCall_HorizontalMove,
    EmergencyStopSignal := ESS,
    Direction := Direction,
    Sensor_01 := LightBarrierSensor_01,
    Sensor_02 := LightBarrierSensor_02,
    AutomaticMode := AutomaticMode,
    ResetCall => ResetMethodCall); // AxisControl_MultipleInputSensors
Motor_Control := HRL_CB_HorizontalMove.MotorControl_01;

{attribute 'TcRpcEnable' := '1'}
METHOD Abort : HRESULT
VAR_INPUT
	hdl : UDINT; // Do not change, used by server.
END_VAR
callCounterAbort := callCounterAbort + 1;
END_METHOD

{attribute 'TcRpcEnable' := '1'}
METHOD CheckState : HRESULT
VAR_INPUT
	hdl : UDINT; // Do not change, used by server.
END_VAR
VAR_OUTPUT
	bBusy : BOOL; // Do not change. Used by server to find out if the job is finished
	
	// List of OutputArguments for OPC UA method, may be customized
	State : BOOL; // Abgeschlossener MethodCall
	MethodCall: BOOL; //Input Recall
END_VAR
callCounterCheckState := callCounterCheckState + 1;
IF NOT jobFinished THEN
	bBusy := TRUE; // job is not finished yet
	CheckState := 0; // no error
ELSE
	bBusy := FALSE; // job is finished
	CheckState := 0; // done, no error occured during execution (OPC UA StatusCode "GOOD")
	jobFinished := FALSE;
	State := ResetMethodCall;
	MethodCall := MethodCall_HorizontalMove;
END_IF
END_METHOD

{attribute 'TcRpcEnable' := '1'}
METHOD Start : HRESULT
VAR_INPUT
	// List of InputArguments for OPC UA method, may be customized
	MethodCall : BOOL; // some description
	MovementDirection : BOOL;	
END_VAR
VAR_OUTPUT
	hdl : UDINT; // Do not change, used by server.
END_VAR
callCounterStart := callCounterStart + 1;

MethodCall_HorizontalMove := MethodCall;
MovementDirection := Direction;

jobRunning := TRUE;
Start := 0; // no error occured, e.g. while parsing the input arguments (0 = OPC UA StatusCode "GOOD")
END_METHOD

END_FUNCTION_BLOCK

// ---- POUs/AtomicSkills/AxisControl_MultipleInputSensors.TcPOU
FUNCTION_BLOCK AxisControl_MultipleInputSensors
VAR_INPUT
	MethodCall: BOOL;
	EmergencyStopSignal : BOOL;
	Direction : BOOL;
	Sensor_01: BOOL;
	Sensor_02: BOOL;
	TouchSensorRelief: BOOL;
	TOF_Time_MotorControl: TIME;
	TOF_Time_TouchSensorRelief: TIME;
	AutomaticMode: BOOL;
END_VAR

VAR_OUTPUT
	MotorControl_01: BOOL;
	MotorControl_02: BOOL;
	ResetCall: BOOL;
END_VAR

VAR
//FlipFlop
	RS_AxisControl: RS;
	RS_TouchSensorRelief: RS;
//Zeitverzögerung
	TOF_TouchSensorRelief: TOF;
	TOF_MotorControl: TOF;	
//Flanke	
	R_TRIG_MethodCall: R_TRIG;
END_VAR
VAR // added by the converter: edge detectors and wires of the graphical bodies
    _w1 : BOOL;
END_VAR

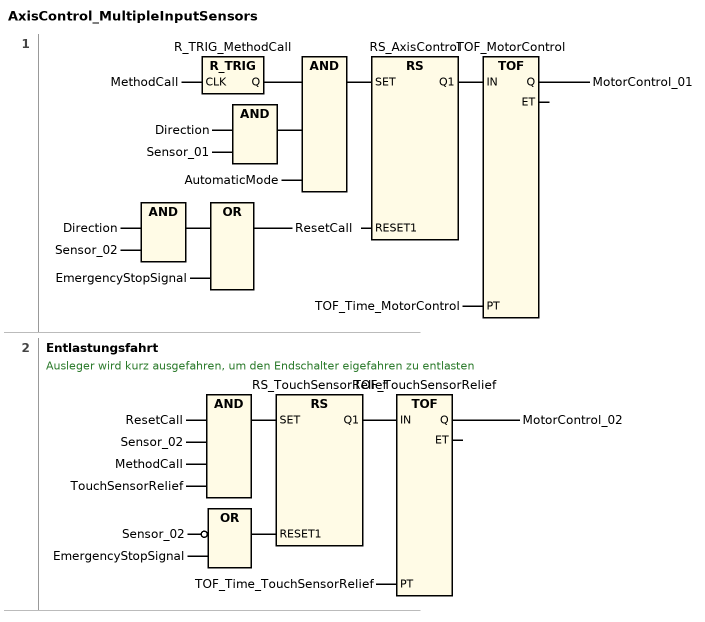
// NETWORK 1
R_TRIG_MethodCall(CLK := MethodCall); // R_TRIG
_w1 := Direction AND Sensor_02 OR EmergencyStopSignal;
ResetCall := _w1;
RS_AxisControl(SET := R_TRIG_MethodCall.Q AND (Direction AND Sensor_01) AND AutomaticMode, RESET1 := _w1); // RS
TOF_MotorControl(IN := RS_AxisControl.Q1, PT := TOF_Time_MotorControl); // TOF
MotorControl_01 := TOF_MotorControl.Q;

// NETWORK 2: Entlastungsfahrt
// Ausleger wird kurz ausgefahren, um den Endschalter eigefahren zu entlasten
RS_TouchSensorRelief(SET := ResetCall AND Sensor_02 AND MethodCall AND TouchSensorRelief, RESET1 := NOT Sensor_02 OR EmergencyStopSignal); // RS
TOF_TouchSensorRelief(IN := RS_TouchSensorRelief.Q1, PT := TOF_Time_TouchSensorRelief); // TOF
MotorControl_02 := TOF_TouchSensorRelief.Q;

END_FUNCTION_BLOCK

// ---- POUs/Moduls/HRL_Skills/HRL_RGB_AS_HorizontalMoveSensors.TcPOU
{attribute 'OPC.UA.DA.JobMethod' := 'JobMethode_HorizontalMove'}
FUNCTION_BLOCK HRL_RGB_AS_HorizontalMoveSensors
VAR
	AlwaysTrue : BOOL := TRUE;
	// Used for debugging purposes to display InputArguments of method call
	MethodCall_HorizontalMove : BOOL := FALSE; // used to store InputArg "MethodCall" from Start() method
	ResetMethodCall	: BOOL := FALSE;	
	Direction : BOOL := FALSE; // defines movement direction
	TSR : BOOL; // Variable that is needed to perform the relief of the touch sensor
	callCounterStart : ULINT; // counts how many times the Start() method has been called
	callCounterCheckState : ULINT; // counts how many times the CheckState() method has been called
	callCounterAbort : ULINT; // counts how many times the Abort() method has been called
	
	// Variables to determine if a job has been started (Start() method has been called) or finished
	jobRunning : BOOL;
	jobFinished : BOOL;

	// State machine variable
	state : UDINT;
	
	// FB Intatziation Variable
	HRL_RGB_HorizontalMove : AxisControl_MultipleInputSensors;
END_VAR
	
VAR_INPUT
	ESS: BOOL;
	TouchSensor_01 : BOOL;
	TouchSensor_02 : BOOL;
	TOF_Time_TSR : TIME;
	AutomaticMode: BOOL;
END_VAR

VAR_OUTPUT
	Motor_Control_01 : BOOL;
	Motor_Control_02 : BOOL;
END_VAR

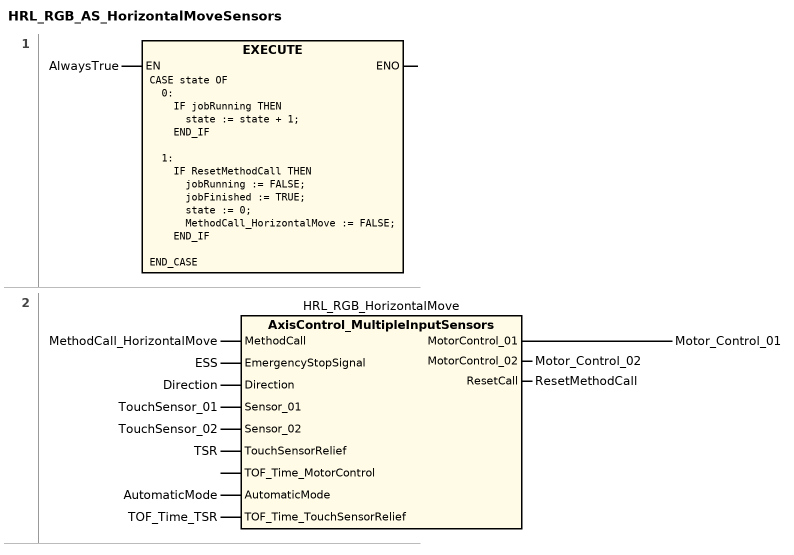
// NETWORK 1
IF AlwaysTrue THEN
    CASE state OF
    	0:
    		IF jobRunning THEN
    			state := state + 1;
    		END_IF
    		
    	1:
    		IF ResetMethodCall THEN
    			jobRunning := FALSE;
    			jobFinished := TRUE;
    			state := 0;
    			MethodCall_HorizontalMove := FALSE;
    		END_IF
    		
    END_CASE
END_IF

// NETWORK 2
HRL_RGB_HorizontalMove(
    MethodCall := MethodCall_HorizontalMove,
    EmergencyStopSignal := ESS,
    Direction := Direction,
    Sensor_01 := TouchSensor_01,
    Sensor_02 := TouchSensor_02,
    TouchSensorRelief := TSR,
    AutomaticMode := AutomaticMode,
    TOF_Time_TouchSensorRelief := TOF_Time_TSR,
    MotorControl_02 => Motor_Control_02,
    ResetCall => ResetMethodCall); // AxisControl_MultipleInputSensors
Motor_Control_01 := HRL_RGB_HorizontalMove.MotorControl_01;

{attribute 'TcRpcEnable' := '1'}
METHOD Abort : HRESULT
VAR_INPUT
	hdl : UDINT; // Do not change, used by server.
END_VAR
callCounterAbort := callCounterAbort + 1;
END_METHOD

{attribute 'TcRpcEnable' := '1'}
METHOD CheckState : HRESULT
VAR_INPUT
	hdl : UDINT; // Do not change, used by server.
END_VAR
VAR_OUTPUT
	bBusy : BOOL; // Do not change. Used by server to find out if the job is finished
	
	// List of OutputArguments for OPC UA method, may be customized
	State : BOOL; // Abgeschlossener MethodCall
	MethodCall: BOOL; //Input Recall
END_VAR
callCounterCheckState := callCounterCheckState + 1;
IF NOT jobFinished THEN
	bBusy := TRUE; // job is not finished yet
	CheckState := 0; // no error
ELSE
	bBusy := FALSE; // job is finished
	CheckState := 0; // done, no error occured during execution (OPC UA StatusCode "GOOD")
	jobFinished := FALSE;
	State := ResetMethodCall;
	MethodCall := MethodCall_HorizontalMove;
END_IF
END_METHOD

{attribute 'TcRpcEnable' := '1'}
METHOD Start : HRESULT
VAR_INPUT
	// List of InputArguments for OPC UA method, may be customized
	MethodCall : BOOL; // some description
	MovementDirection : BOOL;
	EndschalterEntlastung : BOOL;
END_VAR
VAR_OUTPUT
	hdl : UDINT; // Do not change, used by server.
END_VAR
callCounterStart := callCounterStart + 1;

MethodCall_HorizontalMove := MethodCall;
MovementDirection := Direction;
EndschalterEntlastung := EndschalterEntlastung;

jobRunning := TRUE;
Start := 0; // no error occured, e.g. while parsing the input arguments (0 = OPC UA StatusCode "GOOD")
END_METHOD

END_FUNCTION_BLOCK

// ---- POUs/Moduls/HRL_Skills/HRL_RGB_AS_VerticalMoveEncoder.TcPOU
{attribute 'OPC.UA.DA.JobMethod' := 'JobMethode_VerticalMove'}
FUNCTION_BLOCK HRL_RGB_AS_VerticalMoveEncoder
VAR
	AlwaysTrue : BOOL := TRUE;
	// Used for debugging purposes to display InputArguments of method call
	MethodCall_VerticalMove : BOOL := FALSE; // used to store InputArg "MethodCall" from Start() method
	ResetMethodCall	: BOOL := FALSE;
	Direction : BOOL := FALSE;
	EncoderTargetPosition_01 : UDINT;
	EncoderTargetPosition_02 : UDINT;
	TSR : BOOL;
	callCounterStart : ULINT; // counts how many times the Start() method has been called
	callCounterCheckState : ULINT; // counts how many times the CheckState() method has been called
	callCounterAbort : ULINT; // counts how many times the Abort() method has been called
	
	// Variables to determine if a job has been started (Start() method has been called) or finished
	jobRunning : BOOL;
	jobFinished : BOOL;

	// State machine variable
	state : UDINT;
	
	// FB Intatziation Variable
	HRL_RGB_VerticalMoveWithEncoder : AxisControl_Encoder;
END_VAR
	
VAR_INPUT
	ESS: BOOL;
	EncoderStartPosition_01 : UDINT;
	EncoderStartPosition_02 : UDINT;
	TS01 : BOOL;
	TOF_TSR_TIME : TIME;
	AutomaticMode: BOOL;
END_VAR

VAR_OUTPUT
	Motor_Control_01 : BOOL;
	Motor_Control_02 : BOOL;
END_VAR

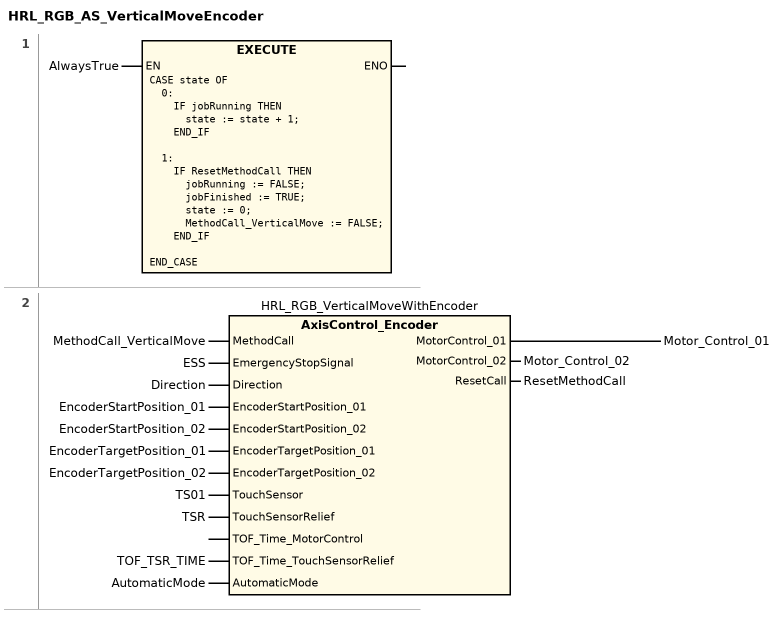
// NETWORK 1
IF AlwaysTrue THEN
    CASE state OF
    	0:
    		IF jobRunning THEN
    			state := state + 1;
    		END_IF
    		
    	1:
    		IF ResetMethodCall THEN
    			jobRunning := FALSE;
    			jobFinished := TRUE;
    			state := 0;
    			MethodCall_VerticalMove := FALSE;
    		END_IF
    		
    END_CASE
END_IF

// NETWORK 2
HRL_RGB_VerticalMoveWithEncoder(
    MethodCall := MethodCall_VerticalMove,
    EmergencyStopSignal := ESS,
    Direction := Direction,
    EncoderStartPosition_01 := EncoderStartPosition_01,
    EncoderStartPosition_02 := EncoderStartPosition_02,
    EncoderTargetPosition_01 := EncoderTargetPosition_01,
    EncoderTargetPosition_02 := EncoderTargetPosition_02,
    TouchSensor := TS01,
    TouchSensorRelief := TSR,
    TOF_Time_TouchSensorRelief := TOF_TSR_TIME,
    AutomaticMode := AutomaticMode,
    MotorControl_02 => Motor_Control_02,
    ResetCall => ResetMethodCall); // AxisControl_Encoder
Motor_Control_01 := HRL_RGB_VerticalMoveWithEncoder.MotorControl_01;

{attribute 'TcRpcEnable' := '1'}
METHOD Abort : HRESULT
VAR_INPUT
	hdl : UDINT; // Do not change, used by server.
END_VAR
callCounterAbort := callCounterAbort + 1;
END_METHOD

{attribute 'TcRpcEnable' := '1'}
METHOD CheckState : HRESULT
VAR_INPUT
	hdl : UDINT; // Do not change, used by server.
END_VAR
VAR_OUTPUT
	bBusy : BOOL; // Do not change. Used by server to find out if the job is finished
	
	// List of OutputArguments for OPC UA method, may be customized
	State : BOOL; // Abgeschlossener MethodCall
	MethodCall: BOOL; //Input Recall
END_VAR
callCounterCheckState := callCounterCheckState + 1;
IF NOT jobFinished THEN
	bBusy := TRUE; // job is not finished yet
	CheckState := 0; // no error
ELSE
	bBusy := FALSE; // job is finished
	CheckState := 0; // done, no error occured during execution (OPC UA StatusCode "GOOD")
	jobFinished := FALSE;
	State := ResetMethodCall;
	MethodCall := MethodCall_VerticalMove;
END_IF
END_METHOD

{attribute 'TcRpcEnable' := '1'}
METHOD Start : HRESULT
VAR_INPUT
	// List of InputArguments for OPC UA method, may be customized
	MethodCall : BOOL; // some description
	MovementDirection : BOOL;
	EncoderPositionVertical_01 : UDINT;
	EncoderPositionVertical_02 : UDINT;
	TouchSensorRelief : BOOL;
END_VAR
VAR_OUTPUT
	hdl : UDINT; // Do not change, used by server.
END_VAR
callCounterStart := callCounterStart + 1;

MethodCall_VerticalMove := MethodCall;
MovementDirection := Direction;
EncoderTargetPosition_01 := EncoderPositionVertical_01;
EncoderTargetPosition_02 := EncoderPositionVertical_02;
TouchSensorRelief := TSR;

jobRunning := TRUE;
Start := 0; // no error occured, e.g. while parsing the input arguments (0 = OPC UA StatusCode "GOOD")
END_METHOD

END_FUNCTION_BLOCK

// ---- POUs/AtomicSkills/AxisControl_Encoder.TcPOU
FUNCTION_BLOCK AxisControl_Encoder
VAR_INPUT
	MethodCall: BOOL;
	EmergencyStopSignal : BOOL;
	Direction : BOOL;
	EncoderStartPosition_01 : UDINT;
	EncoderStartPosition_02 : UDINT;
	EncoderTargetPosition_01 : UDINT;
	EncoderTargetPosition_02 : UDINT;	
	TouchSensor: BOOL;
	TouchSensorRelief : BOOL;
	TOF_Time_MotorControl: TIME;
	TOF_Time_TouchSensorRelief: TIME;
	AutomaticMode: BOOL;
END_VAR

VAR_OUTPUT
	MotorControl_01: BOOL;
	MotorControl_02: BOOL;
	ResetCall: BOOL;
END_VAR

VAR
//FlipFlop
	RS_AxisControl: RS;
	RS_Endschalter_Entlasten: RS;
//Zeitverzögerung
	TOF_Endschalter_Entlasten: TOF;
	TOF_MotorControl: TOF;	
//Flanke	
	R_TRIG_MethodCall: R_TRIG;
	R_TRIG_EncoderPos_01 : R_TRIG;
	R_TRIG_EncoderPos_02 : R_TRIG;

END_VAR
VAR // added by the converter: edge detectors and wires of the graphical bodies
    _w1, _w2 : BOOL;
END_VAR

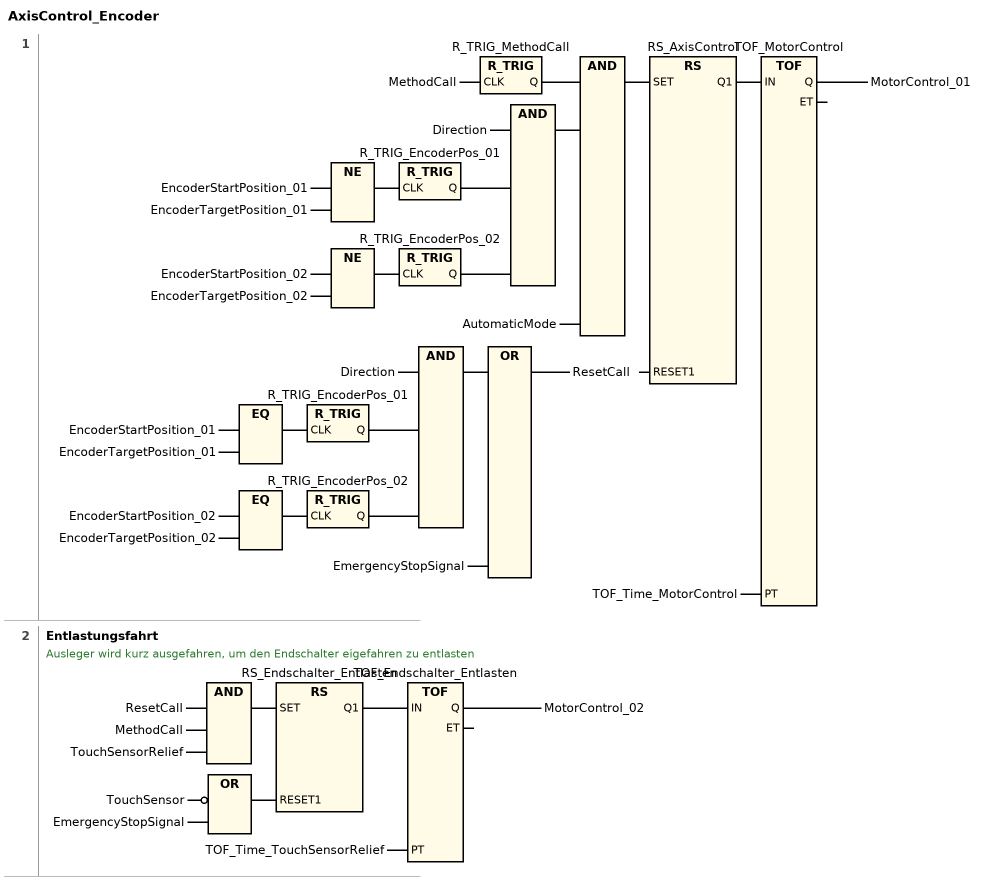
// NETWORK 1
R_TRIG_MethodCall(CLK := MethodCall); // R_TRIG
R_TRIG_EncoderPos_01(CLK := EncoderStartPosition_01 <> EncoderTargetPosition_01); // R_TRIG
R_TRIG_EncoderPos_02(CLK := EncoderStartPosition_02 <> EncoderTargetPosition_02); // R_TRIG
_w2 := R_TRIG_MethodCall.Q AND (Direction AND R_TRIG_EncoderPos_01.Q AND R_TRIG_EncoderPos_02.Q) AND AutomaticMode;
R_TRIG_EncoderPos_01(CLK := EncoderStartPosition_01 = EncoderTargetPosition_01); // R_TRIG
R_TRIG_EncoderPos_02(CLK := EncoderStartPosition_02 = EncoderTargetPosition_02); // R_TRIG
_w1 := Direction AND R_TRIG_EncoderPos_01.Q AND R_TRIG_EncoderPos_02.Q OR EmergencyStopSignal;
ResetCall := _w1;
RS_AxisControl(SET := _w2, RESET1 := _w1); // RS
TOF_MotorControl(IN := RS_AxisControl.Q1, PT := TOF_Time_MotorControl); // TOF
MotorControl_01 := TOF_MotorControl.Q;

// NETWORK 2: Entlastungsfahrt
// Ausleger wird kurz ausgefahren, um den Endschalter eigefahren zu entlasten
RS_Endschalter_Entlasten(SET := ResetCall AND MethodCall AND TouchSensorRelief, RESET1 := NOT TouchSensor OR EmergencyStopSignal); // RS
TOF_Endschalter_Entlasten(IN := RS_Endschalter_Entlasten.Q1, PT := TOF_Time_TouchSensorRelief); // TOF
MotorControl_02 := TOF_Endschalter_Entlasten.Q;

END_FUNCTION_BLOCK

// ---- POUs/Moduls/HRL_Skills/HRL_RGB_AS_HorizontalMoveEncoder.TcPOU
{attribute 'OPC.UA.DA.JobMethod' := 'JobMethode_HorizontalMove'}
FUNCTION_BLOCK HRL_RGB_AS_HorizontalMoveEncoder
VAR
	AlwaysTrue : BOOL := TRUE;
	// Used for debugging purposes to display InputArguments of method call
	MethodCall_HorizontalMove : BOOL := FALSE; // used to store InputArg "MethodCall" from Start() method
	ResetMethodCall	: BOOL := FALSE;	
	Direction : BOOL := FALSE;
	EncoderTargetPosition_01 : UDINT;
	EncoderTargetPosition_02 : UDINT;
	TSR: BOOL;
	callCounterStart : ULINT; // counts how many times the Start() method has been called
	callCounterCheckState : ULINT; // counts how many times the CheckState() method has been called
	callCounterAbort : ULINT; // counts how many times the Abort() method has been called
	
	// Variables to determine if a job has been started (Start() method has been called) or finished
	jobRunning : BOOL;
	jobFinished : BOOL;

	// State machine variable
	state : UDINT;
	
	// FB Intatziation Variable
	HRL_RGB_HorizontalMoveWithEncoder : AxisControl_Encoder;
END_VAR
	
VAR_INPUT
	ESS: BOOL;
	EncoderStartPosition_01 : UDINT;
	EncoderStartPosition_02 : UDINT;
	TS01 : BOOL;
	TOF_Time_TSR : TIME;
	AutomaticMode: BOOL;
END_VAR

VAR_OUTPUT
	Motor_Control_01 : BOOL;
	Motor_Control_02 : BOOL;
END_VAR

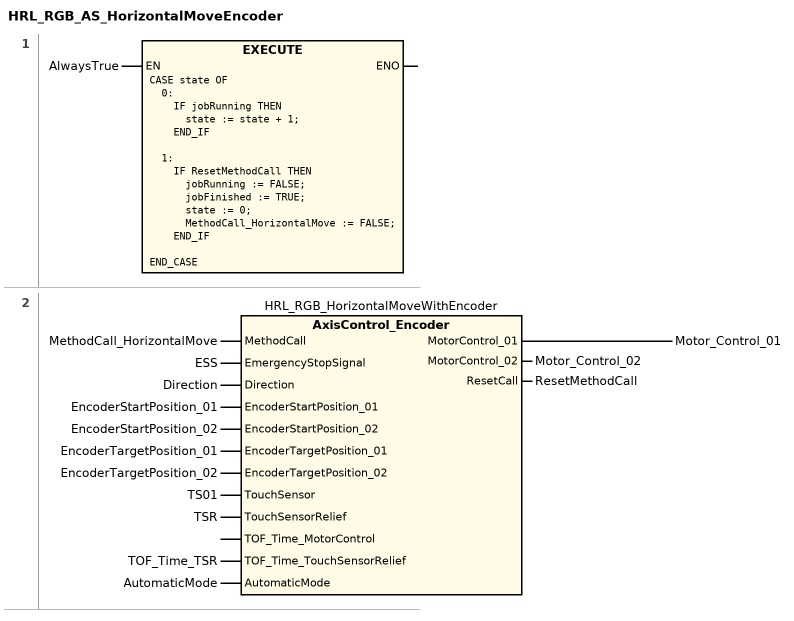
// NETWORK 1
IF AlwaysTrue THEN
    CASE state OF
    	0:
    		IF jobRunning THEN
    			state := state + 1;
    		END_IF
    		
    	1:
    		IF ResetMethodCall THEN
    			jobRunning := FALSE;
    			jobFinished := TRUE;
    			state := 0;
    			MethodCall_HorizontalMove := FALSE;
    		END_IF
    		
    END_CASE
END_IF

// NETWORK 2
HRL_RGB_HorizontalMoveWithEncoder(
    MethodCall := MethodCall_HorizontalMove,
    EmergencyStopSignal := ESS,
    Direction := Direction,
    EncoderStartPosition_01 := EncoderStartPosition_01,
    EncoderStartPosition_02 := EncoderStartPosition_02,
    EncoderTargetPosition_01 := EncoderTargetPosition_01,
    EncoderTargetPosition_02 := EncoderTargetPosition_02,
    TouchSensor := TS01,
    TouchSensorRelief := TSR,
    TOF_Time_TouchSensorRelief := TOF_Time_TSR,
    AutomaticMode := AutomaticMode,
    MotorControl_02 => Motor_Control_02,
    ResetCall => ResetMethodCall); // AxisControl_Encoder
Motor_Control_01 := HRL_RGB_HorizontalMoveWithEncoder.MotorControl_01;

{attribute 'TcRpcEnable' := '1'}
METHOD Abort : HRESULT
VAR_INPUT
	hdl : UDINT; // Do not change, used by server.
END_VAR
callCounterAbort := callCounterAbort + 1;
END_METHOD

{attribute 'TcRpcEnable' := '1'}
METHOD CheckState : HRESULT
VAR_INPUT
	hdl : UDINT; // Do not change, used by server.
END_VAR
VAR_OUTPUT
	bBusy : BOOL; // Do not change. Used by server to find out if the job is finished
	
	// List of OutputArguments for OPC UA method, may be customized
	State : BOOL; // Abgeschlossener MethodCall
	MethodCall: BOOL; //Input Recall
END_VAR
callCounterCheckState := callCounterCheckState + 1;
IF NOT jobFinished THEN
	bBusy := TRUE; // job is not finished yet
	CheckState := 0; // no error
ELSE
	bBusy := FALSE; // job is finished
	CheckState := 0; // done, no error occured during execution (OPC UA StatusCode "GOOD")
	jobFinished := FALSE;
	State := ResetMethodCall;
	MethodCall := MethodCall_HorizontalMove;
END_IF
END_METHOD

{attribute 'TcRpcEnable' := '1'}
METHOD Start : HRESULT
VAR_INPUT
	// List of InputArguments for OPC UA method, may be customized
	MethodCall : BOOL; // some description
	MovementDirection : BOOL;
	EncoderPositionHorizontal_01 : UDINT;
	EncoderPositionHorizontal_02 : UDINT;
	TouchSensorRelief : BOOL;
END_VAR
VAR_OUTPUT
	hdl : UDINT; // Do not change, used by server.
END_VAR
callCounterStart := callCounterStart + 1;

MethodCall_HorizontalMove := MethodCall;
MovementDirection := Direction;
EncoderTargetPosition_01 := EncoderPositionHorizontal_01;
EncoderTargetPosition_02 := EncoderPositionHorizontal_02;
TouchSensorRelief := TSR;

jobRunning := TRUE;
Start := 0; // no error occured, e.g. while parsing the input arguments (0 = OPC UA StatusCode "GOOD")
END_METHOD

END_FUNCTION_BLOCK

// ---- POUs/ControlOfOutputs/HRL_ControlOfOutputs.TcPOU
FUNCTION_BLOCK HRL_ControlOfOutputs
VAR_INPUT
	F4				: BOOL;
	F1				: BOOL;
	A2				: BOOL;
	A1				: BOOL;
	Start			: BOOL;
	CB_forwards 	: BOOL; //GVL_HRL.HRL_MOT_Foerderband_vorwaerts
	CB_backwards 	: BOOL; //GVL_HRL.HRL_MOT_Foerderband_rueckwaerts
	RGB_Forwards01 : BOOL; //GVL_HRL.HRL_MOT_Ausleger_vorwaerts
	RGB_Backwards02 : BOOL; //GVL_HRL.HRL_MOT_Ausleger_vorwaerts
	RGB_Forwards02 : BOOL; //GVL_HRL.HRL_MOT_Ausleger_rueckwaerts
	RGB_Backwards01 : BOOL; //GVL_HRL.HRL_MOT_Ausleger_rueckwaerts
	RGB_VertikalDown01 : BOOL; //GVL_HRL.HRL_MOT_vertikal_runter
	RGB_VertikalUp02 : BOOL; //GVL_HRL.HRL_MOT_vertikal_runter
	RGB_VertikalDown02 : BOOL; //GVL_HRL.HRL_MOT_vertikal_hoch
	RGB_VertikalUp01 : BOOL; //GVL_HRL.HRL_MOT_vertikal_hoch
	RGB_HorizontalForwards01 : BOOL; //GVL_HRL.HRL_MOT_horizontal_zum_Regal
	RGB_HorizontalBackwards02 : BOOL; //GVL_HRL.HRL_MOT_horizontal_zum_Regal
	RGB_HorizontalForwards02 : BOOL; //GVL_HRL.HRL_MOT_horizontal_zum_Foerderband
	RGB_HorizontalBackwards01 : BOOL; //GVL_HRL.HRL_MOT_horizontal_zum_Foerderband
END_VAR
VAR_OUTPUT
	ConveyorBeltForward: BOOL;
	ConveyorBeltBackward: BOOL;
	RGB_Forwards: BOOL;
	RGB_Backwards: BOOL;
	RGB_VerticalDown: BOOL;
	RGB_VerticalUp: BOOL;
	RGB_HorizontalForward: BOOL;
	RGB_HorizontalBackward: BOOL;
	Light_Q1: BOOL;
	Light_Q2: BOOL;
	Light_Q3: BOOL;
END_VAR
VAR
END_VAR

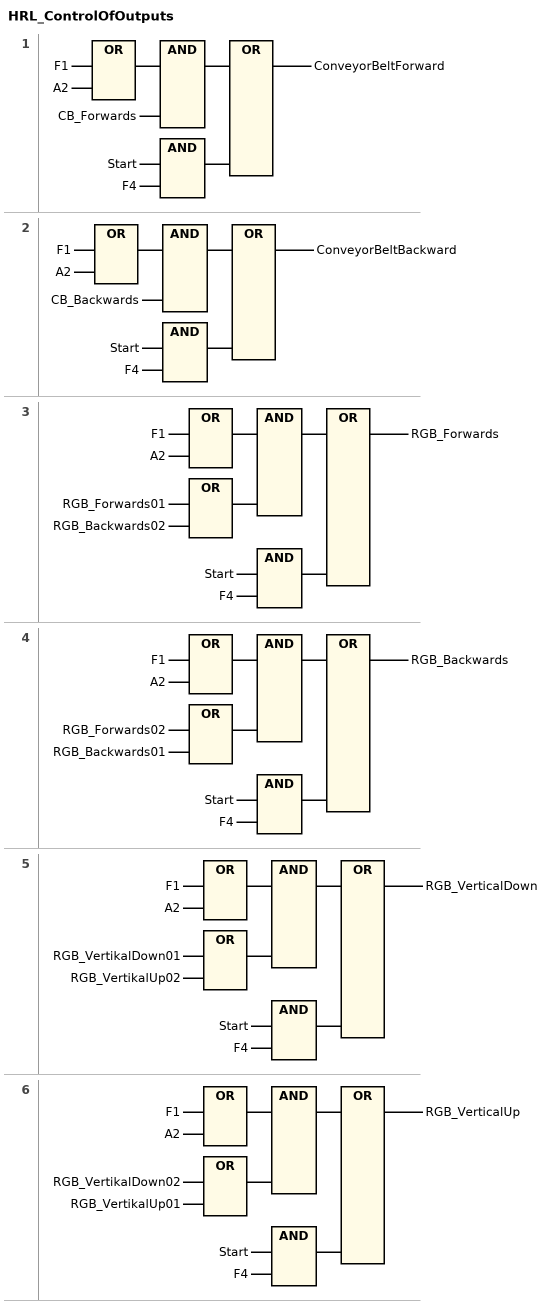
// NETWORK 1
ConveyorBeltForward := (F1 OR A2) AND CB_Forwards OR Start AND F4;

// NETWORK 2
ConveyorBeltBackward := (F1 OR A2) AND CB_Backwards OR Start AND F4;

// NETWORK 3
RGB_Forwards := (F1 OR A2) AND (RGB_Forwards01 OR RGB_Backwards02) OR Start AND F4;

// NETWORK 4
RGB_Backwards := (F1 OR A2) AND (RGB_Forwards02 OR RGB_Backwards01) OR Start AND F4;

// NETWORK 5
RGB_VerticalDown := (F1 OR A2) AND (RGB_VertikalDown01 OR RGB_VertikalUp02) OR Start AND F4;

// NETWORK 6
RGB_VerticalUp := (F1 OR A2) AND (RGB_VertikalDown02 OR RGB_VertikalUp01) OR Start AND F4;

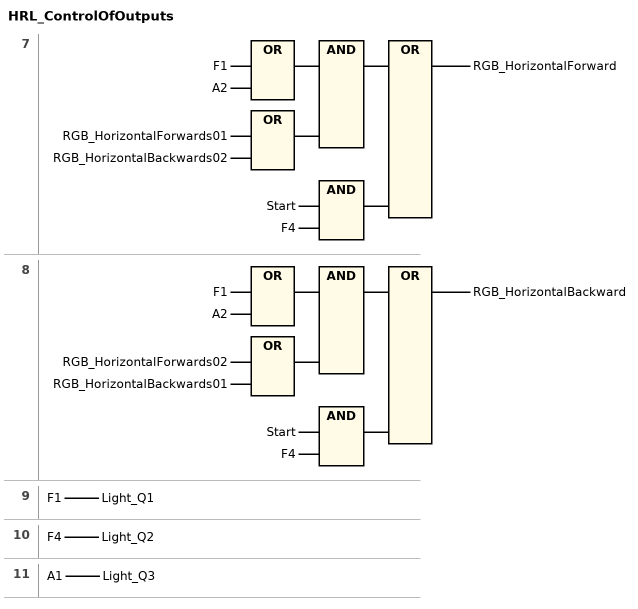
// NETWORK 7
RGB_HorizontalForward := (F1 OR A2) AND (RGB_HorizontalForwards01 OR RGB_HorizontalBackwards02) OR Start AND F4;

// NETWORK 8
RGB_HorizontalBackward := (F1 OR A2) AND (RGB_HorizontalForwards02 OR RGB_HorizontalBackwards01) OR Start AND F4;

// NETWORK 9
Light_Q1 := F1;

// NETWORK 10
Light_Q2 := F4;

// NETWORK 11
Light_Q3 := A1;

END_FUNCTION_BLOCK

// ---- POUs/OperatingModes/HRL_OperatingModes.TcPOU
FUNCTION_BLOCK HRL_OperatingModes
VAR_INPUT
	Start 			: BOOL;
	Stop			: BOOL;
	Reset			: BOOL;
	Schalter		: BOOL;
	Schrittkette_GS : BOOL;
END_VAR
VAR_OUTPUT
	A1 : BOOL; //Initialzustand
	A2 : BOOL; //Stillstand angefordert am Ende des Zyklus
//	A3 : BOOL; //Stillstand angefordert in einem bestimmten Zustand
//	A4 : BOOL; //Erhaltener Stillstand
//	A5 : BOOL; //Vorbereitung zur Wiederaufnahme nach Störung
	A6 : BOOL; //Fahrt in den Initialzustand
	F1 : BOOL; //Normalbetrieb
//	F2 : BOOL; //Anfahren
//	F3 : BOOL; //Abfahren
	F4 : BOOL; //Handbetrieb
//	F5 : BOOL; //Schrittbetrieb
//	F6 : BOOL; //Testbetrieb
//	D1 : BOOL; //Not-Aus
//	D2 : BOOL; //DIagnose und Störbehandlung
//	D3 : BOOL; //Produktion trotz Störung
END_VAR
VAR
	bFirstScan : BOOL := TRUE;	

	RS_InitialState: RS;	
	RS_InitialDrive: RS;
	RS_ManualOperationMode: RS;
	RS_AutomaticOperationMode: RS;
	RS_CycleEnded: RS;

	R_TRIG_Manual: R_TRIG;
	R_TRIG_Automatic: R_TRIG;
	R_TRIG_InitialDrive: R_TRIG;
	R_TRIG_CycleEnded: R_TRIG;
	R_TRIG_Init: R_TRIG;
END_VAR
VAR // added by the converter: edge detectors and wires of the graphical bodies
    _w1 : BOOL;
END_VAR

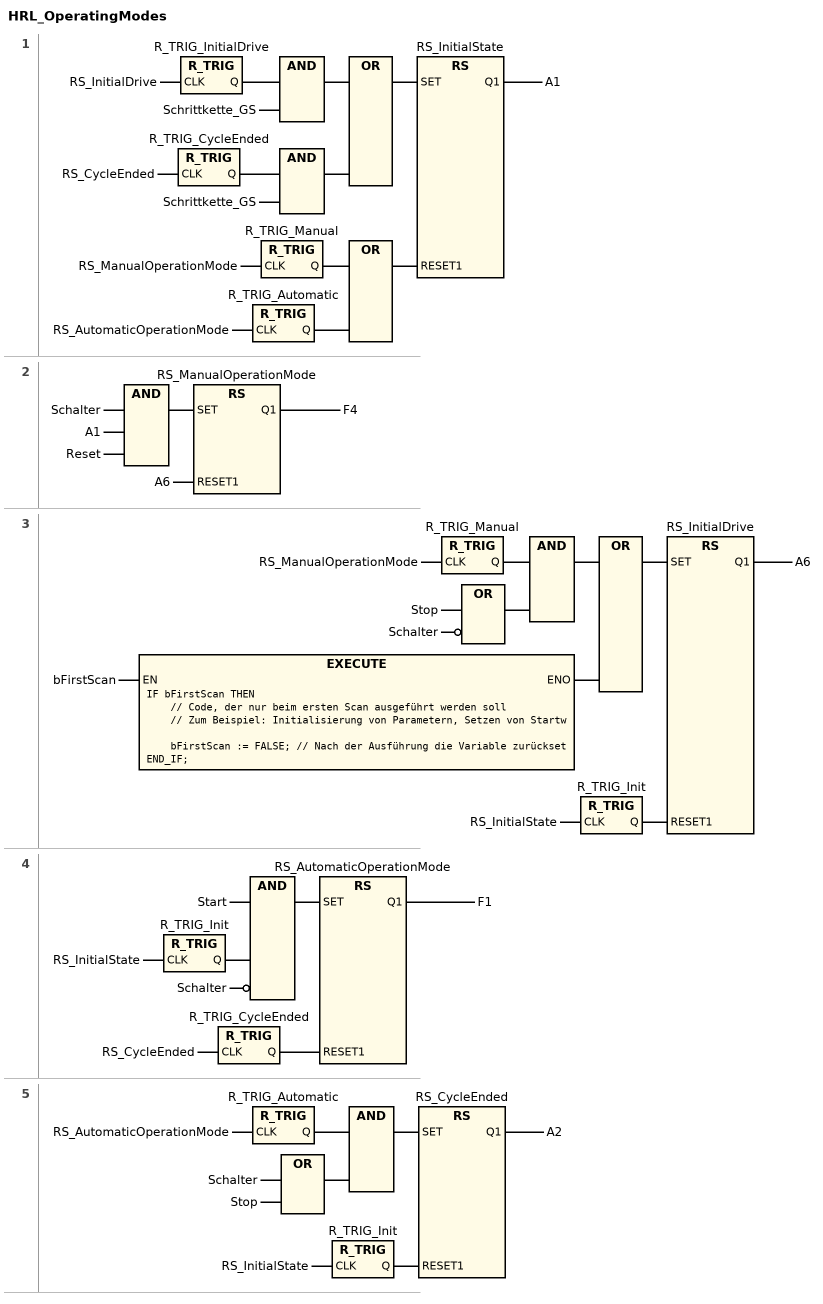
// NETWORK 1
R_TRIG_InitialDrive(CLK := RS_InitialDrive); // R_TRIG
R_TRIG_CycleEnded(CLK := RS_CycleEnded); // R_TRIG
R_TRIG_Manual(CLK := RS_ManualOperationMode); // R_TRIG
R_TRIG_Automatic(CLK := RS_AutomaticOperationMode); // R_TRIG
RS_InitialState(SET := R_TRIG_InitialDrive.Q AND Schrittkette_GS OR R_TRIG_CycleEnded.Q AND Schrittkette_GS, RESET1 := R_TRIG_Manual.Q OR R_TRIG_Automatic.Q); // RS
A1 := RS_InitialState.Q1;

// NETWORK 2
RS_ManualOperationMode(SET := Schalter AND A1 AND Reset, RESET1 := A6); // RS
F4 := RS_ManualOperationMode.Q1;

// NETWORK 3
R_TRIG_Manual(CLK := RS_ManualOperationMode); // R_TRIG
_w1 := bFirstScan;
IF _w1 THEN
    IF bFirstScan THEN
        // Code, der nur beim ersten Scan ausgeführt werden soll
        // Zum Beispiel: Initialisierung von Parametern, Setzen von Startwerten etc.
    	
        bFirstScan := FALSE; // Nach der Ausführung die Variable zurücksetzen
    END_IF;
END_IF
R_TRIG_Init(CLK := RS_InitialState); // R_TRIG
RS_InitialDrive(SET := R_TRIG_Manual.Q AND (Stop OR NOT Schalter) OR _w1, RESET1 := R_TRIG_Init.Q); // RS
A6 := RS_InitialDrive.Q1;

// NETWORK 4
R_TRIG_Init(CLK := RS_InitialState); // R_TRIG
R_TRIG_CycleEnded(CLK := RS_CycleEnded); // R_TRIG
RS_AutomaticOperationMode(SET := Start AND R_TRIG_Init.Q AND NOT Schalter, RESET1 := R_TRIG_CycleEnded.Q); // RS
F1 := RS_AutomaticOperationMode.Q1;

// NETWORK 5
R_TRIG_Automatic(CLK := RS_AutomaticOperationMode); // R_TRIG
R_TRIG_Init(CLK := RS_InitialState); // R_TRIG
RS_CycleEnded(SET := R_TRIG_Automatic.Q AND (Schalter OR Stop), RESET1 := R_TRIG_Init.Q); // RS
A2 := RS_CycleEnded.Q1;

END_FUNCTION_BLOCK

// ---- POUs/MethodenBeispiele/HRL_NMethod_Auslagern.TcPOU
FUNCTION_BLOCK PUBLIC HRL_NMethod_Auslagern
VAR_INPUT
	NotAusSignal: BOOL;
	LS01_Start: BOOL;
	LS02_Ende: BOOL;
END_VAR
VAR_OUTPUT
	Motor_Auslagern: BOOL;
	Status: BOOL;
END_VAR
VAR
	Transport_Auslagern: Transport_Unidirectional;
	Input_C: BOOL;
	R_TRIG: R_TRIG;
END_VAR

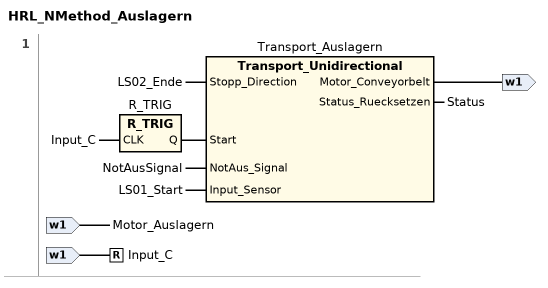
// NETWORK 1
R_TRIG(CLK := Input_C);
Transport_Auslagern(
    Stopp_Direction := LS02_Ende,
    Start := R_TRIG.Q,
    NotAus_Signal := NotAusSignal,
    Input_Sensor := LS01_Start,
    Status_Ruecksetzen => Status); // Transport_Unidirectional
Motor_Auslagern := Transport_Auslagern.Motor_Conveyorbelt;
Input_C R= Transport_Auslagern.Motor_Conveyorbelt;

{attribute 'TcRpcEnable' := '1'}
METHOD METH_Auslagern : BOOL
VAR_INPUT
	MethodCall_C : BOOL;
END_VAR
Input_C := MethodCall_C;
END_METHOD

END_FUNCTION_BLOCK

// ---- POUs/AtomicSkills/Auto_ColorDetection.TcPOU
FUNCTION_BLOCK Auto_ColorDetection
VAR_INPUT
	ColorSensor: INT;
	ColorCode_1: INT;
	ColorCode_2: INT;
	ColorCode_3: INT;
END_VAR
VAR_OUTPUT
	Color_1: BOOL;
	Color_2: BOOL;
	Color_3: BOOL;
END_VAR
VAR

END_VAR

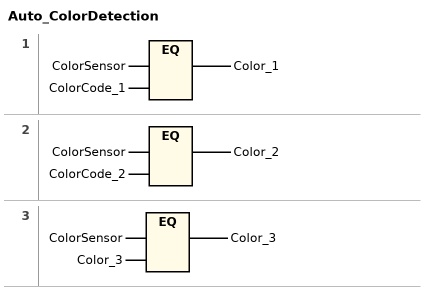
// NETWORK 1
Color_1 := ColorSensor = ColorCode_1;

// NETWORK 2
Color_2 := ColorSensor = ColorCode_2;

// NETWORK 3
Color_3 := ColorSensor = Color_3;

END_FUNCTION_BLOCK

// ---- POUs/AtomicSkills/CompressorControl.TcPOU
FUNCTION_BLOCK CompressorControl
VAR_INPUT
	MethodCall: BOOL;
	NotAus_Signal : BOOL;
	Destination : BOOL;
	LightSensor_01: BOOL;
	LightSensor_02: BOOL;
	TS_Endschalter_01: BOOL;
	TS_Endschalter_02: BOOL;
	EncoderStartPosition_01 : BOOL;
	EncoderStartPosition_02 : BOOL;
	EncoderStartPosition_03 : BOOL;
	EncoderStartPosition_04 : BOOL;
	EncoderStartPosition_05 : BOOL;
	EncoderStartPosition_06 : BOOL;
	EncoderTargetPosition_01 : BOOL;
	EncoderTargetPosition_02 : BOOL;
	EncoderTargetPosition_03 : BOOL;
	EncoderTargetPosition_04 : BOOL;
	EncoderTargetPosition_05 : BOOL;
	EncoderTargetPosition_06 : BOOL;	
	PowerOnDelay_Kompressor: TIME;
	PowerOnDelay_Ventil: TIME;
	AutomaticMode: BOOL;
END_VAR
VAR_OUTPUT
	Ansteuerung_Compressor : BOOL;
	Ansteuerung_Ventil : BOOL;
END_VAR
VAR
//FlipFlop
	RS_Vakuumkompressor: RS;
	RS_Vakuumventil: RS;
//Zeitverzögerung
	TON_Ansteuerung_Kompressor: TON;
	TON_Ansteuerung_Ventil: TON;
//Flanke	
	R_TRIG_MethodCall: R_TRIG;
END_VAR

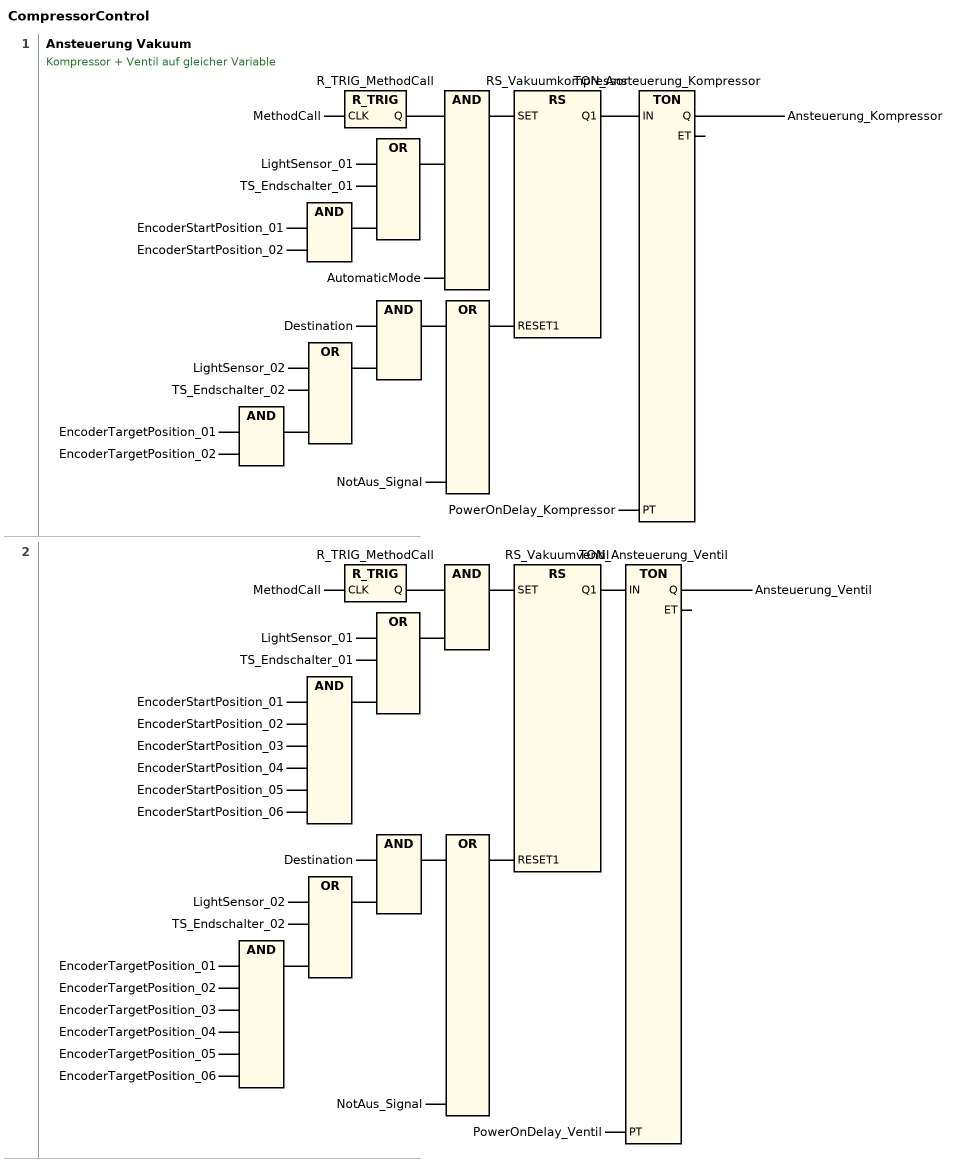
// NETWORK 1: Ansteuerung Vakuum
// Kompressor + Ventil auf gleicher Variable
R_TRIG_MethodCall(CLK := MethodCall); // R_TRIG
RS_Vakuumkompressor(SET := R_TRIG_MethodCall.Q AND (LightSensor_01 OR TS_Endschalter_01 OR EncoderStartPosition_01 AND EncoderStartPosition_02) AND AutomaticMode, RESET1 := Destination AND (LightSensor_02 OR TS_Endschalter_02 OR EncoderTargetPosition_01 AND EncoderTargetPosition_02) OR NotAus_Signal); // RS
TON_Ansteuerung_Kompressor(IN := RS_Vakuumkompressor.Q1, PT := PowerOnDelay_Kompressor); // TON
Ansteuerung_Kompressor := TON_Ansteuerung_Kompressor.Q;

// NETWORK 2
R_TRIG_MethodCall(CLK := MethodCall); // R_TRIG
RS_Vakuumventil(SET := R_TRIG_MethodCall.Q AND (LightSensor_01 OR TS_Endschalter_01 OR EncoderStartPosition_01 AND EncoderStartPosition_02 AND EncoderStartPosition_03 AND EncoderStartPosition_04 AND EncoderStartPosition_05 AND EncoderStartPosition_06), RESET1 := Destination AND (LightSensor_02 OR TS_Endschalter_02 OR EncoderTargetPosition_01 AND EncoderTargetPosition_02 AND EncoderTargetPosition_03 AND EncoderTargetPosition_04 AND EncoderTargetPosition_05 AND EncoderTargetPosition_06) OR NotAus_Signal); // RS
TON_Ansteuerung_Ventil(IN := RS_Vakuumventil.Q1, PT := PowerOnDelay_Ventil); // TON
Ansteuerung_Ventil := TON_Ansteuerung_Ventil.Q;

END_FUNCTION_BLOCK

// ---- POUs/AtomicSkills/SecuringWorkpiece.TcPOU
FUNCTION_BLOCK SecuringWorkpiece
VAR_INPUT
	MethodCall : BOOL;
	TS_Endschalter_01: BOOL;
	TS_Endschalter_02: BOOL;
	SecuringTime : TIME;
	NotAusSignal : BOOL;
	AutomaticMode: BOOL;
END_VAR
VAR_OUTPUT
	SecuringProcess : BOOL;
END_VAR
VAR
//FlipFlop
	RS_SecuringProcessON: RS;	
//Zeitverzögerung
	TON_SecuringTime: TON;
//Flanke	
	R_TRIG_MethodCall: R_TRIG;
END_VAR

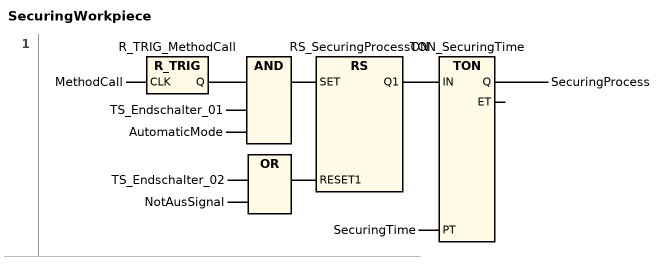
// NETWORK 1
R_TRIG_MethodCall(CLK := MethodCall); // R_TRIG
RS_SecuringProcessON(SET := R_TRIG_MethodCall.Q AND TS_Endschalter_01 AND AutomaticMode, RESET1 := TS_Endschalter_02 OR NotAusSignal); // RS
TON_SecuringTime(IN := RS_SecuringProcessON.Q1, PT := SecuringTime); // TON
SecuringProcess := TON_SecuringTime.Q;

END_FUNCTION_BLOCK

// ---- POUs/AtomicSkills/StampingProcess.TcPOU
FUNCTION_BLOCK StampingProcess
VAR_INPUT
	MethodCall : BOOL;
	InputSensor: BOOL;
	StampingTime : TIME;
	NotAusSignal : BOOL;
	AutomaticMode: BOOL;
END_VAR
VAR_OUTPUT
	StampingProcess : BOOL;
END_VAR
VAR
//FlipFlop
	RS_StampingProcess: RS;
//Zeitverzögerung
	TOF_StampingTime: TOF;
//Flanke	
	R_TRIG_MethodCall: R_TRIG;
END_VAR
VAR // added by the converter: edge detectors and wires of the graphical bodies
    _w1 : BOOL;
END_VAR

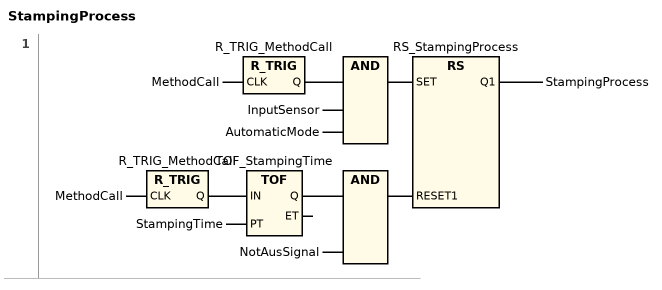
// NETWORK 1
R_TRIG_MethodCall(CLK := MethodCall); // R_TRIG
_w1 := R_TRIG_MethodCall.Q AND InputSensor AND AutomaticMode;
R_TRIG_MethodCall(CLK := MethodCall); // R_TRIG
TOF_StampingTime(IN := R_TRIG_MethodCall.Q, PT := StampingTime); // TOF
RS_StampingProcess(SET := _w1, RESET1 := TOF_StampingTime.Q AND NotAusSignal); // RS
StampingProcess := RS_StampingProcess.Q1;

END_FUNCTION_BLOCK

// ---- POUs/AtomicSkills/HardeningProcess.TcPOU
FUNCTION_BLOCK HardeningProcess
VAR_INPUT
	MethodCall : BOOL;
	InputSensor: BOOL;
	HardeningTime : TIME;
	NotAusSignal : BOOL;
	AutomaticMode: BOOL;
END_VAR
VAR_OUTPUT
	HardeningProcess : BOOL;
END_VAR
VAR
//FlipFlop
	RS_HardeningProcess: RS;
//Zeitverzögerung
	TOF_HardeningTime: TOF;
//Flanke	
	R_TRIG_MethodCall: R_TRIG;
END_VAR
VAR // added by the converter: edge detectors and wires of the graphical bodies
    _w1 : BOOL;
END_VAR

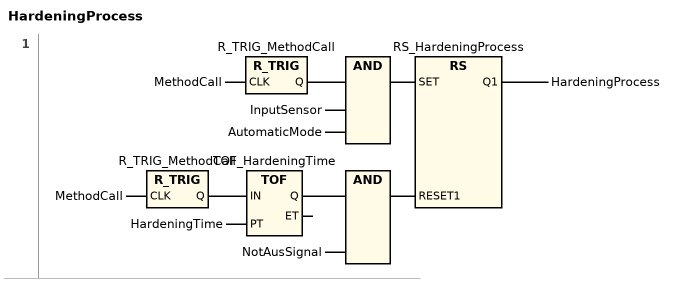
// NETWORK 1
R_TRIG_MethodCall(CLK := MethodCall); // R_TRIG
_w1 := R_TRIG_MethodCall.Q AND InputSensor AND AutomaticMode;
R_TRIG_MethodCall(CLK := MethodCall); // R_TRIG
TOF_HardeningTime(IN := R_TRIG_MethodCall.Q, PT := HardeningTime); // TOF
RS_HardeningProcess(SET := _w1, RESET1 := TOF_HardeningTime.Q AND NotAusSignal); // RS
HardeningProcess := RS_HardeningProcess.Q1;

END_FUNCTION_BLOCK

// ---- POUs/AtomicSkills/CuttingProcess.TcPOU
FUNCTION_BLOCK CuttingProcess
VAR_INPUT
	MethodCall : BOOL;
	InputSensor: BOOL;
	CuttingTime : TIME;
	NotAusSignal : BOOL;
	AutomaticMode: BOOL;
END_VAR
VAR_OUTPUT
	CuttingProcess : BOOL;
END_VAR
VAR
//FlipFlop
	RS_CuttingProcess: RS;
//Zeitverzögerung
	TOF_CuttingTime: TOF;
//Flanke	
	R_TRIG_MethodCall: R_TRIG;
END_VAR
VAR // added by the converter: edge detectors and wires of the graphical bodies
    _w1 : BOOL;
END_VAR

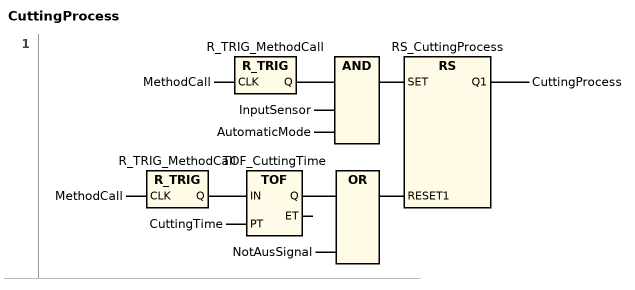
// NETWORK 1
R_TRIG_MethodCall(CLK := MethodCall); // R_TRIG
_w1 := R_TRIG_MethodCall.Q AND InputSensor AND AutomaticMode;
R_TRIG_MethodCall(CLK := MethodCall); // R_TRIG
TOF_CuttingTime(IN := R_TRIG_MethodCall.Q, PT := CuttingTime); // TOF
RS_CuttingProcess(SET := _w1, RESET1 := TOF_CuttingTime.Q OR NotAusSignal); // RS
CuttingProcess := RS_CuttingProcess.Q1;

END_FUNCTION_BLOCK

// ---- POUs/ControlOfOutputs/MBS_ControlOfOutputs.TcPOU
FUNCTION_BLOCK MBS_ControlOfOutputs
VAR_INPUT
END_VAR
VAR_OUTPUT
END_VAR
VAR
END_VAR

// NETWORK 1

END_FUNCTION_BLOCK

// ---- POUs/ControlOfOutputs/SST_ControlOfOutputs.TcPOU
FUNCTION_BLOCK SST_ControlOfOutputs
VAR_INPUT
END_VAR
VAR_OUTPUT
END_VAR
VAR
END_VAR

// NETWORK 1

END_FUNCTION_BLOCK

// ---- POUs/ControlOfOutputs/VSG_ControlOfOutputs.TcPOU
FUNCTION_BLOCK VSG_ControlOfOutputs
VAR_INPUT
END_VAR
VAR_OUTPUT
END_VAR
VAR
END_VAR

// NETWORK 1

END_FUNCTION_BLOCK

// ---- POUs/MethodenBeispiele/FB_MyOpcUaMethod.TcPOU
FUNCTION_BLOCK PUBLIC FB_MyOpcUaMethod
VAR_INPUT
	in1 : INT;
	in2 : INT;
END_VAR
VAR_OUTPUT
	result : INT;
END_VAR

{attribute 'TcRpcEnable' := '1'}
METHOD PUBLIC Multiply : INT
VAR_INPUT
	a : INT;
	b : INT;
END_VAR
Multiply := a * b;
END_METHOD

END_FUNCTION_BLOCK

// ---- POUs/MethodenBeispiele/JobMethode_Schablone.TcPOU
{attribute 'OPC.UA.DA.JobMethod' := 'JobMethode_Schablone'}
FUNCTION_BLOCK JobMethode_Schablone
VAR
	AlwaysTrue : BOOL := TRUE;
	// Used for debugging purposes to display InputArguments of method call
	MethodCall_Name : BOOL := FALSE; // used to store InputArg "MethodCall" from Start() method
	Direction_01 : BOOL := FALSE;
	Direction_02 : BOOL := FALSE;
	TS_EndschalterEntlastung : BOOL;
	callCounterStart : ULINT; // counts how many times the Start() method has been called
	callCounterCheckState : ULINT; // counts how many times the CheckState() method has been called
	callCounterAbort : ULINT; // counts how many times the Abort() method has been called
	
	// Variables to determine if a job has been started (Start() method has been called) or finished
	jobRunning : BOOL;
	jobFinished : BOOL;

	// State machine variable
	state : UDINT;
	
	//Variablen des Transport FBs
	ResetCall : BOOL := FALSE;	
	JobMethode_Name : AxisControl_MultipleInputSensors;
END_VAR
	
VAR_INPUT
	NotAusSignal: BOOL;
	LightSensor_01 : BOOL;
	LightSensor_02 : BOOL;
	TS_Endschalter_01 : BOOL;
	TS_Endschalter_02 : BOOL;
	TOF_Time_Motoransteuerung : TIME;
	TOF_Time_EndschalterEntlastung : TIME;
END_VAR

VAR_OUTPUT
	Motor_Ansteuerung01 : BOOL;
	Motor_Ansteuerung02 : BOOL;
END_VAR

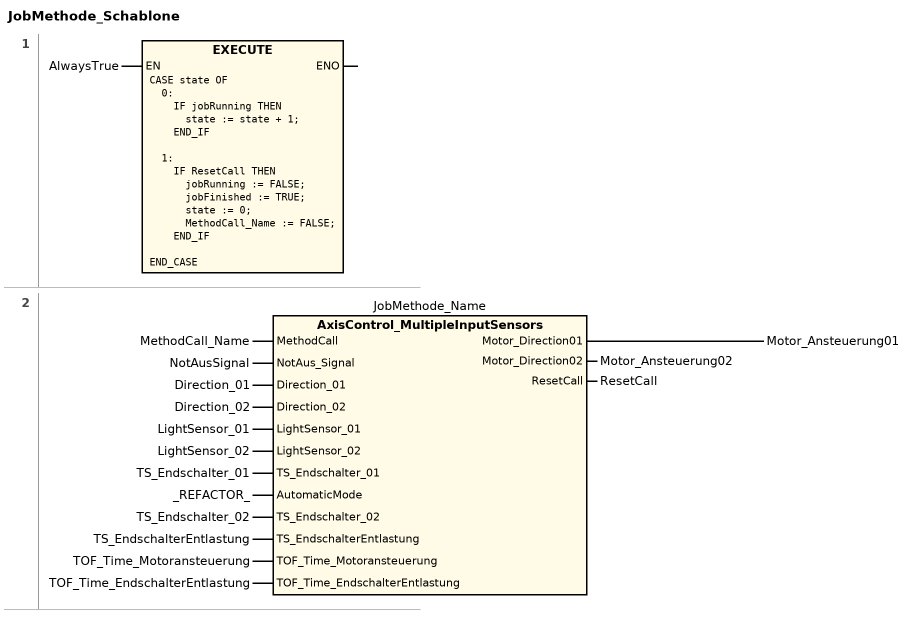
// NETWORK 1
IF AlwaysTrue THEN
    CASE state OF
    	0:
    		IF jobRunning THEN
    			state := state + 1;
    		END_IF
    		
    	1:
    		IF ResetCall THEN
    			jobRunning := FALSE;
    			jobFinished := TRUE;
    			state := 0;
    			MethodCall_Name := FALSE;
    		END_IF
    		
    END_CASE
END_IF

// NETWORK 2
JobMethode_Name(
    MethodCall := MethodCall_Name,
    NotAus_Signal := NotAusSignal,
    Direction_01 := Direction_01,
    Direction_02 := Direction_02,
    LightSensor_01 := LightSensor_01,
    LightSensor_02 := LightSensor_02,
    TS_Endschalter_01 := TS_Endschalter_01,
    AutomaticMode := _REFACTOR_,
    TS_Endschalter_02 := TS_Endschalter_02,
    TS_EndschalterEntlastung := TS_EndschalterEntlastung,
    TOF_Time_Motoransteuerung := TOF_Time_Motoransteuerung,
    TOF_Time_EndschalterEntlastung := TOF_Time_EndschalterEntlastung,
    Motor_Direction02 => Motor_Ansteuerung02,
    ResetCall => ResetCall); // AxisControl_MultipleInputSensors
Motor_Ansteuerung01 := JobMethode_Name.Motor_Direction01;

{attribute 'TcRpcEnable' := '1'}
METHOD Abort : HRESULT
VAR_INPUT
	hdl : UDINT; // Do not change, used by server.
END_VAR
callCounterAbort := callCounterAbort + 1;
END_METHOD

{attribute 'TcRpcEnable' := '1'}
METHOD CheckState : HRESULT
VAR_INPUT
	hdl : UDINT; // Do not change, used by server.
END_VAR
VAR_OUTPUT
	bBusy : BOOL; // Do not change. Used by server to find out if the job is finished
	
	// List of OutputArguments for OPC UA method, may be customized
	State : BOOL; // Abgeschlossener MethodCall
	MethodCall: BOOL; //Input Recall
END_VAR
callCounterCheckState := callCounterCheckState + 1;
IF NOT jobFinished THEN
	bBusy := TRUE; // job is not finished yet
	CheckState := 0; // no error
ELSE
	bBusy := FALSE; // job is finished
	CheckState := 0; // done, no error occured during execution (OPC UA StatusCode "GOOD")
	jobFinished := FALSE;
	State := ResetCall;
	MethodCall := MethodCall_Name;
END_IF
END_METHOD

{attribute 'TcRpcEnable' := '1'}
METHOD Start : HRESULT
VAR_INPUT
	// List of InputArguments for OPC UA method, may be customized
	MethodCall : BOOL; // some description
	DirectionPointA : BOOL;
	DirectionPointB : BOOL;
	EndschalterEntlastung : BOOL;	
END_VAR
VAR_OUTPUT
	hdl : UDINT; // Do not change, used by server.
END_VAR
callCounterStart := callCounterStart + 1;

MethodCall_Name := MethodCall;
DirectionPointA := Direction_01;
DirectionPointB := Direction_02;
EndschalterEntlastung := EndschalterEntlastung;

IF DirectionPointA := TRUE THEN
	DirectionPointB := FALSE;
END_IF

IF DirectionPointB := TRUE THEN
	DirectionPointA := FALSE;
END_IF

jobRunning := TRUE;
Start := 0; // no error occured, e.g. while parsing the input arguments (0 = OPC UA StatusCode "GOOD")
END_METHOD

END_FUNCTION_BLOCK

// ---- POUs/MethodenBeispiele/JobMethode.TcPOU
{attribute 'OPC.UA.DA.JobMethod' := 'MyJob'}
FUNCTION_BLOCK JobMethode
VAR
	// Used for debugging purposes to display InputArguments of method call
	Input_a : INT; // used to store InputArg "a" from Start() method
	Input_b : LREAL; // used to store InputArg "b" from Start() method
	Input_c : BOOL; // used to store InputArg "c" from Start() method
//	Input_d : ST_Complex_1; // used to store InputArg "d" from Start() method
	callCounterStart : ULINT; // counts how many times the Start() method has been called
	callCounterCheckState : ULINT; // counts how many times the CheckState() method has been called
	callCounterAbort : ULINT; // counts how many times the Abort() method has been called
	
	// Timer to "artificially delay" job execution
	timer : TON := (PT:=T#4S);
	
	// Variables to determine if a job has been started (Start() method has been called) or finished
	jobRunning : BOOL;
	jobFinished : BOOL;

	// State machine variable
	state : UDINT;
END_VAR

CASE state OF
	0:
		IF jobRunning THEN
			state := state + 1;
		END_IF
		
	1:
		timer(IN:=TRUE);
		IF timer.Q THEN
			timer(IN:=FALSE);
			jobRunning := FALSE;
			jobFinished := TRUE;
			state := 0;
		END_IF
		
END_CASE

{attribute 'TcRpcEnable' := '1'}
METHOD Abort : HRESULT
VAR_INPUT
	hdl : UDINT; // Do not change, used by server.
END_VAR
callCounterAbort := callCounterAbort + 1;
END_METHOD

{attribute 'TcRpcEnable' := '1'}
METHOD CheckState : HRESULT
VAR_INPUT
	hdl : UDINT; // Do not change, used by server.
END_VAR
VAR_OUTPUT
	bBusy : BOOL; // Do not change. Used by server to find out if the job is finished
	
	// List of OutputArguments for OPC UA method, may be customized
	a : INT; // some description
	b : LREAL; // some description
	c : BOOL; // some description
//	d : ST_Complex_1; // some description
END_VAR
callCounterCheckState := callCounterCheckState + 1;
IF NOT jobFinished THEN
	bBusy := TRUE; // job is not finished yet
	CheckState := 0; // no error
ELSE
	bBusy := FALSE; // job is finished
	CheckState := 0; // done, no error occured during execution (OPC UA StatusCode "GOOD")
	jobFinished := FALSE;
	a := Input_a;
	b := Input_b;
	c := Input_c;
//	d := Input_d;
END_IF
END_METHOD

{attribute 'TcRpcEnable' := '1'}
METHOD Start : HRESULT
VAR_INPUT
	// List of InputArguments for OPC UA method, may be customized
	a : INT; // some description
	b : LREAL; // some description
	c : BOOL; // some description
//	d : ST_Complex_1; // some description
END_VAR
VAR_OUTPUT
	hdl : UDINT; // Do not change, used by server.
END_VAR
callCounterStart := callCounterStart + 1;
Input_a := a;
Input_b := b;
Input_c := c;
//Input_d := d;
jobRunning := TRUE;
Start := 0; // no error occured, e.g. while parsing the input arguments (0 = OPC UA StatusCode "GOOD")
END_METHOD

END_FUNCTION_BLOCK

// ---- POUs/Moduls/HRL_Skills/HRL_RGB_InitalStateDrive.TcPOU
FUNCTION_BLOCK HRL_RGB_InitalStateDrive
VAR_INPUT
END_VAR
VAR_OUTPUT
END_VAR
VAR
	HRL_RGB_SRM_InitDrive: AxisControl_MultipleInputSensors;
END_VAR

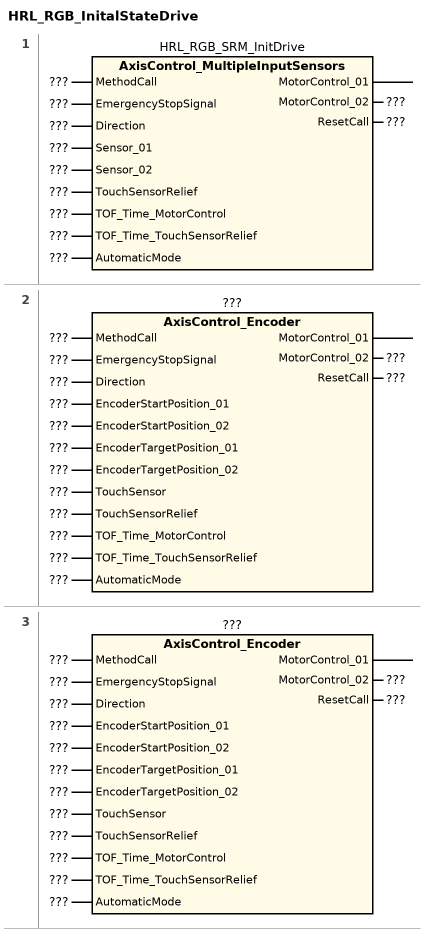
// NETWORK 1
HRL_RGB_SRM_InitDrive(); // AxisControl_MultipleInputSensors

// NETWORK 2
???(); // AxisControl_Encoder

// NETWORK 3
???(); // AxisControl_Encoder

END_FUNCTION_BLOCK

// ---- POUs/Moduls/MBS_Skills/MBS_MR01_AS_HardeningProcess.TcPOU
{attribute 'OPC.UA.DA.JobMethod' := 'JobMethode_HardeningProcess'}
FUNCTION_BLOCK MBS_MR01_AS_HardeningProcess
VAR
	AlwaysTrue : BOOL := TRUE;
	// Used for debugging purposes to display InputArguments of method call
	MethodCall_HardeningProcess : BOOL := FALSE; // used to store InputArg "MethodCall" from Start() method
	ProcessingTime_HardeningProcess : TIME;
	TS_EndschalterEntlastung : BOOL;
	callCounterStart : ULINT; // counts how many times the Start() method has been called
	callCounterCheckState : ULINT; // counts how many times the CheckState() method has been called
	callCounterAbort : ULINT; // counts how many times the Abort() method has been called
	
	// Variables to determine if a job has been started (Start() method has been called) or finished
	jobRunning : BOOL;
	jobFinished : BOOL;

	// State machine variable
	state : UDINT;
	
	//Variablen des FBs
	ResetCall : BOOL;
	MBS_MR01_HardeningProcess : HardeningProcess;
END_VAR
	
VAR_INPUT
	NotAusSignal: BOOL;
	LightSensor_01 : BOOL;
END_VAR

VAR_OUTPUT
	Oven_Ansteuerung : BOOL;
END_VAR

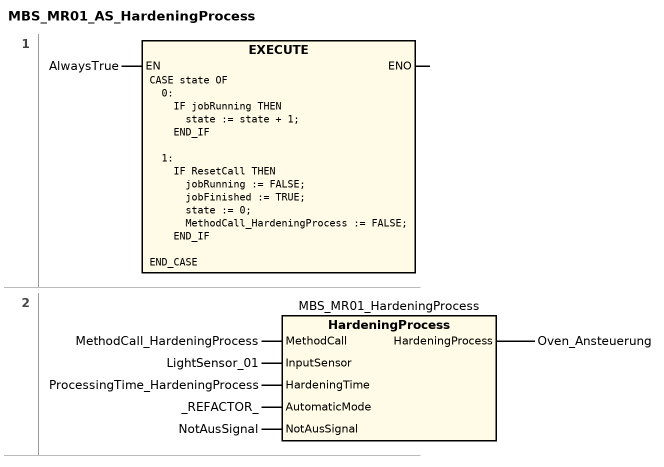
// NETWORK 1
IF AlwaysTrue THEN
    CASE state OF
    	0:
    		IF jobRunning THEN
    			state := state + 1;
    		END_IF
    		
    	1:
    		IF ResetCall THEN
    			jobRunning := FALSE;
    			jobFinished := TRUE;
    			state := 0;
    			MethodCall_HardeningProcess := FALSE;
    		END_IF
    		
    END_CASE
END_IF

// NETWORK 2
MBS_MR01_HardeningProcess(
    MethodCall := MethodCall_HardeningProcess,
    InputSensor := LightSensor_01,
    HardeningTime := ProcessingTime_HardeningProcess,
    AutomaticMode := _REFACTOR_,
    NotAusSignal := NotAusSignal); // HardeningProcess
Oven_Ansteuerung := MBS_MR01_HardeningProcess.HardeningProcess;

{attribute 'TcRpcEnable' := '1'}
METHOD Abort : HRESULT
VAR_INPUT
	hdl : UDINT; // Do not change, used by server.
END_VAR
callCounterAbort := callCounterAbort + 1;
END_METHOD

{attribute 'TcRpcEnable' := '1'}
METHOD CheckState : HRESULT
VAR_INPUT
	hdl : UDINT; // Do not change, used by server.
END_VAR
VAR_OUTPUT
	bBusy : BOOL; // Do not change. Used by server to find out if the job is finished
	
	// List of OutputArguments for OPC UA method, may be customized
	State : BOOL; // Abgeschlossener MethodCall
	MethodCall: BOOL; //Input Recall
END_VAR
callCounterCheckState := callCounterCheckState + 1;
IF NOT jobFinished THEN
	bBusy := TRUE; // job is not finished yet
	CheckState := 0; // no error
ELSE
	bBusy := FALSE; // job is finished
	CheckState := 0; // done, no error occured during execution (OPC UA StatusCode "GOOD")
	jobFinished := FALSE;
	State := ResetCall;
	MethodCall := MethodCall_HardeningProcess;
END_IF
END_METHOD

{attribute 'TcRpcEnable' := '1'}
METHOD Start : HRESULT
VAR_INPUT
	// List of InputArguments for OPC UA method, may be customized
	MethodCall : BOOL; // some description
	ProcessingTime : TIME;
END_VAR
VAR_OUTPUT
	hdl : UDINT; // Do not change, used by server.
END_VAR
callCounterStart := callCounterStart + 1;

MethodCall_HardeningProcess := MethodCall;
ProcessingTime_HardeningProcess := ProcessingTime;

jobRunning := TRUE;
Start := 0; // no error occured, e.g. while parsing the input arguments (0 = OPC UA StatusCode "GOOD")
END_METHOD

END_FUNCTION_BLOCK

// ---- POUs/Moduls/MBS_Skills/MBS_MR01_AS_SecuringProcess.TcPOU
{attribute 'OPC.UA.DA.JobMethod' := 'JobMethode_SecuringProcess'}
FUNCTION_BLOCK MBS_MR01_AS_SecuringProcess
VAR
	AlwaysTrue : BOOL := TRUE;
	// Used for debugging purposes to display InputArguments of method call
	MethodCall_SecuringProcess : BOOL := FALSE; // used to store InputArg "MethodCall" from Start() method
	ProcessingTime_SecuringProcess : TIME;
	TS_EndschalterEntlastung : BOOL;
	callCounterStart : ULINT; // counts how many times the Start() method has been called
	callCounterCheckState : ULINT; // counts how many times the CheckState() method has been called
	callCounterAbort : ULINT; // counts how many times the Abort() method has been called
	
	// Variables to determine if a job has been started (Start() method has been called) or finished
	jobRunning : BOOL;
	jobFinished : BOOL;

	// State machine variable
	state : UDINT;
	
	//Variablen des FBs
	ResetCall : BOOL;
	MBS_MR01_SecuringProcess : SecuringWorkpiece;
END_VAR
	
VAR_INPUT
	NotAusSignal: BOOL;
	TS_Endschalter_01: BOOL;
	TS_Endschalter_02: BOOL;
END_VAR

VAR_OUTPUT
	SecuringProcess : BOOL;
END_VAR

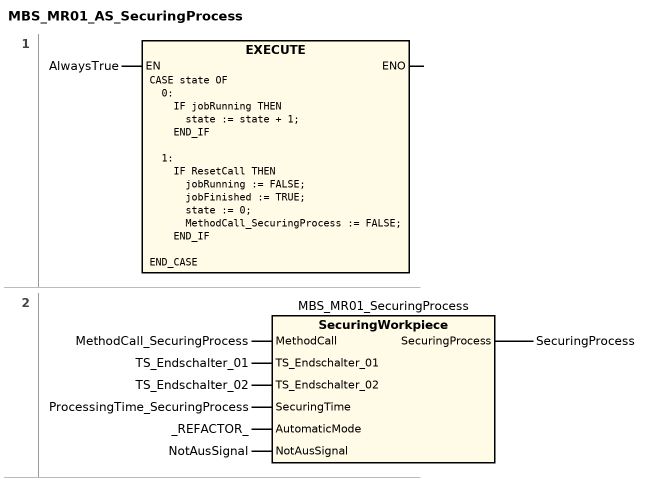
// NETWORK 1
IF AlwaysTrue THEN
    CASE state OF
    	0:
    		IF jobRunning THEN
    			state := state + 1;
    		END_IF
    		
    	1:
    		IF ResetCall THEN
    			jobRunning := FALSE;
    			jobFinished := TRUE;
    			state := 0;
    			MethodCall_SecuringProcess := FALSE;
    		END_IF
    		
    END_CASE
END_IF

// NETWORK 2
MBS_MR01_SecuringProcess(
    MethodCall := MethodCall_SecuringProcess,
    TS_Endschalter_01 := TS_Endschalter_01,
    TS_Endschalter_02 := TS_Endschalter_02,
    SecuringTime := ProcessingTime_SecuringProcess,
    AutomaticMode := _REFACTOR_,
    NotAusSignal := NotAusSignal); // SecuringWorkpiece
SecuringProcess := MBS_MR01_SecuringProcess.SecuringProcess;

{attribute 'TcRpcEnable' := '1'}
METHOD Abort : HRESULT
VAR_INPUT
	hdl : UDINT; // Do not change, used by server.
END_VAR
callCounterAbort := callCounterAbort + 1;
END_METHOD

{attribute 'TcRpcEnable' := '1'}
METHOD CheckState : HRESULT
VAR_INPUT
	hdl : UDINT; // Do not change, used by server.
END_VAR
VAR_OUTPUT
	bBusy : BOOL; // Do not change. Used by server to find out if the job is finished
	
	// List of OutputArguments for OPC UA method, may be customized
	State : BOOL; // Abgeschlossener MethodCall
	MethodCall: BOOL; //Input Recall
END_VAR
callCounterCheckState := callCounterCheckState + 1;
IF NOT jobFinished THEN
	bBusy := TRUE; // job is not finished yet
	CheckState := 0; // no error
ELSE
	bBusy := FALSE; // job is finished
	CheckState := 0; // done, no error occured during execution (OPC UA StatusCode "GOOD")
	jobFinished := FALSE;
	State := ResetCall;
	MethodCall := MethodCall_SecuringProcess;
END_IF
END_METHOD

{attribute 'TcRpcEnable' := '1'}
METHOD Start : HRESULT
VAR_INPUT
	// List of InputArguments for OPC UA method, may be customized
	MethodCall : BOOL; // some description
	ProcessingTime : TIME;
END_VAR
VAR_OUTPUT
	hdl : UDINT; // Do not change, used by server.
END_VAR
callCounterStart := callCounterStart + 1;

MethodCall_SecuringProcess := MethodCall;
ProcessingTime_SecuringProcess := ProcessingTime;

jobRunning := TRUE;
Start := 0; // no error occured, e.g. while parsing the input arguments (0 = OPC UA StatusCode "GOOD")
END_METHOD

END_FUNCTION_BLOCK

// ---- POUs/Moduls/MBS_Skills/MBS_VSG_AS_VerticalMove.TcPOU
{attribute 'OPC.UA.DA.JobMethod' := 'JobMethode_CompressorControl'}
FUNCTION_BLOCK MBS_VSG_AS_VerticalMove
VAR
	AlwaysTrue : BOOL := TRUE;
	// Used for debugging purposes to display InputArguments of method call
	MethodCall_CompressorControl : BOOL := FALSE; // used to store InputArg "MethodCall" from Start() method
	Destination : BOOL;
	TS_EndschalterEntlastung : BOOL;
	callCounterStart : ULINT; // counts how many times the Start() method has been called
	callCounterCheckState : ULINT; // counts how many times the CheckState() method has been called
	callCounterAbort : ULINT; // counts how many times the Abort() method has been called
	
	// Variables to determine if a job has been started (Start() method has been called) or finished
	jobRunning : BOOL;
	jobFinished : BOOL;

	// State machine variable
	state : UDINT;
	
	//Variablen des Transport FBs
	ResetCall : BOOL := FALSE;	
	MBS_VSG_VerticalMove : CompressorControl;
END_VAR
	
VAR_INPUT
	NotAusSignal: BOOL;
//	LightSensor_01 : BOOL;
//	LightSensor_02 : BOOL;
	TS_Endschalter_01 : BOOL;
	TS_Endschalter_02 : BOOL;
	PowerOnDelay_Compressor : TIME;
	PowerOnDelay_Ventil : TIME;
END_VAR

VAR_OUTPUT
	Compressor : BOOL;
	Ventil : BOOL;
END_VAR

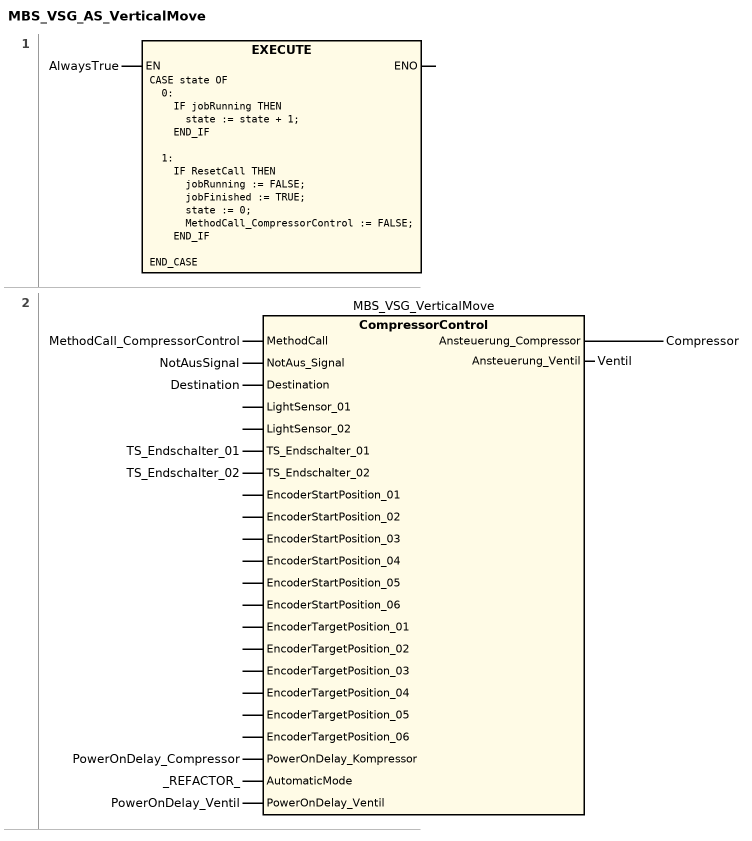
// NETWORK 1
IF AlwaysTrue THEN
    CASE state OF
    	0:
    		IF jobRunning THEN
    			state := state + 1;
    		END_IF
    		
    	1:
    		IF ResetCall THEN
    			jobRunning := FALSE;
    			jobFinished := TRUE;
    			state := 0;
    			MethodCall_CompressorControl := FALSE;
    		END_IF
    		
    END_CASE
END_IF

// NETWORK 2
MBS_VSG_VerticalMove(
    MethodCall := MethodCall_CompressorControl,
    NotAus_Signal := NotAusSignal,
    Destination := Destination,
    TS_Endschalter_01 := TS_Endschalter_01,
    TS_Endschalter_02 := TS_Endschalter_02,
    PowerOnDelay_Kompressor := PowerOnDelay_Compressor,
    AutomaticMode := _REFACTOR_,
    PowerOnDelay_Ventil := PowerOnDelay_Ventil,
    Ansteuerung_Ventil => Ventil); // CompressorControl
Compressor := MBS_VSG_VerticalMove.Ansteuerung_Compressor;

{attribute 'TcRpcEnable' := '1'}
METHOD Abort : HRESULT
VAR_INPUT
	hdl : UDINT; // Do not change, used by server.
END_VAR
callCounterAbort := callCounterAbort + 1;
END_METHOD

{attribute 'TcRpcEnable' := '1'}
METHOD CheckState : HRESULT
VAR_INPUT
	hdl : UDINT; // Do not change, used by server.
END_VAR
VAR_OUTPUT
	bBusy : BOOL; // Do not change. Used by server to find out if the job is finished
	
	// List of OutputArguments for OPC UA method, may be customized
	State : BOOL; // Abgeschlossener MethodCall
	MethodCall: BOOL; //Input Recall
END_VAR
callCounterCheckState := callCounterCheckState + 1;
IF NOT jobFinished THEN
	bBusy := TRUE; // job is not finished yet
	CheckState := 0; // no error
ELSE
	bBusy := FALSE; // job is finished
	CheckState := 0; // done, no error occured during execution (OPC UA StatusCode "GOOD")
	jobFinished := FALSE;
	State := ResetCall;
	MethodCall := MethodCall_CompressorControl;
END_IF
END_METHOD

{attribute 'TcRpcEnable' := '1'}
METHOD Start : HRESULT
VAR_INPUT
	// List of InputArguments for OPC UA method, may be customized
	MethodCall : BOOL; // some description
	Destination : BOOL;	
END_VAR
VAR_OUTPUT
	hdl : UDINT; // Do not change, used by server.
END_VAR
callCounterStart := callCounterStart + 1;

MethodCall_CompressorControl := MethodCall;
Destination := Destination;

jobRunning := TRUE;
Start := 0; // no error occured, e.g. while parsing the input arguments (0 = OPC UA StatusCode "GOOD")
END_METHOD

END_FUNCTION_BLOCK

// ---- POUs/Moduls/MBS_Skills/MBS_MR01_AS_HorizontalMove.TcPOU
{attribute 'OPC.UA.DA.JobMethod' := 'JobMethode_HorizontalMove'}
FUNCTION_BLOCK MBS_MR01_AS_HorizontalMove
VAR
	AlwaysTrue : BOOL := TRUE;
	// Used for debugging purposes to display InputArguments of method call
	MethodCall_HorizontalMove : BOOL := FALSE; // used to store InputArg "MethodCall" from Start() method
	Direction : BOOL := FALSE;
	TS_EndschalterEntlastung : BOOL;
	callCounterStart : ULINT; // counts how many times the Start() method has been called
	callCounterCheckState : ULINT; // counts how many times the CheckState() method has been called
	callCounterAbort : ULINT; // counts how many times the Abort() method has been called
	
	// Variables to determine if a job has been started (Start() method has been called) or finished
	jobRunning : BOOL;
	jobFinished : BOOL;

	// State machine variable
	state : UDINT;
	
	//Variablen des Transport FBs
	ResetCall : BOOL := FALSE;	
	MBS_MR01_HorizontalMove : AxisControl_MultipleInputSensors;
END_VAR
	
VAR_INPUT
	NotAusSignal: BOOL;
	LightSensor_01 : BOOL;
	LightSensor_02 : BOOL;
	TS_Endschalter_01 : BOOL;
	TS_Endschalter_02 : BOOL;
	TOF_Time_Motoransteuerung : TIME;
	TOF_Time_EndschalterEntlastung : TIME;
END_VAR

VAR_OUTPUT
	Motor_Ansteuerung01 : BOOL;
	Motor_Ansteuerung02 : BOOL;
END_VAR

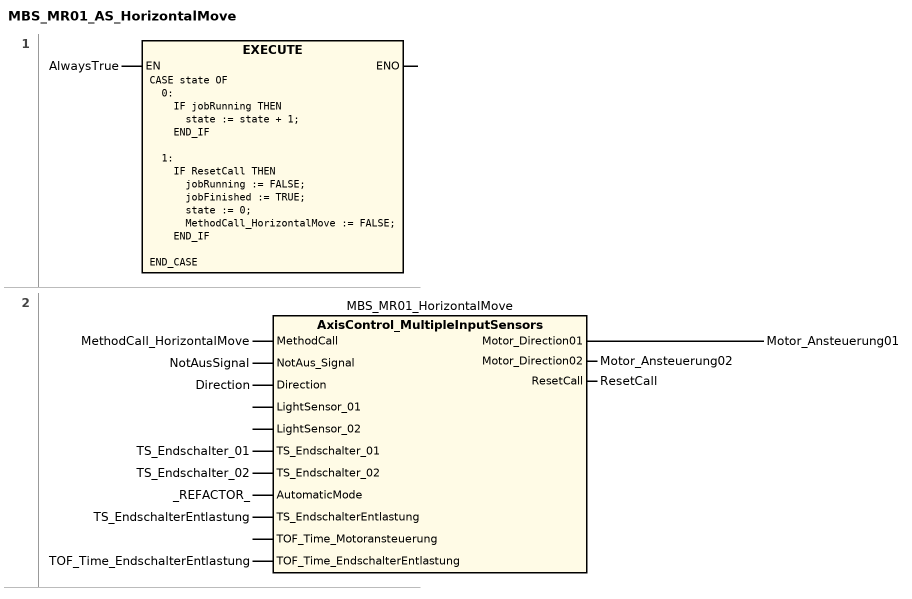
// NETWORK 1
IF AlwaysTrue THEN
    CASE state OF
    	0:
    		IF jobRunning THEN
    			state := state + 1;
    		END_IF
    		
    	1:
    		IF ResetCall THEN
    			jobRunning := FALSE;
    			jobFinished := TRUE;
    			state := 0;
    			MethodCall_HorizontalMove := FALSE;
    		END_IF
    		
    END_CASE
END_IF

// NETWORK 2
MBS_MR01_HorizontalMove(
    MethodCall := MethodCall_HorizontalMove,
    NotAus_Signal := NotAusSignal,
    Direction := Direction,
    TS_Endschalter_01 := TS_Endschalter_01,
    TS_Endschalter_02 := TS_Endschalter_02,
    AutomaticMode := _REFACTOR_,
    TS_EndschalterEntlastung := TS_EndschalterEntlastung,
    TOF_Time_EndschalterEntlastung := TOF_Time_EndschalterEntlastung,
    Motor_Direction02 => Motor_Ansteuerung02,
    ResetCall => ResetCall); // AxisControl_MultipleInputSensors
Motor_Ansteuerung01 := MBS_MR01_HorizontalMove.Motor_Direction01;

{attribute 'TcRpcEnable' := '1'}
METHOD Abort : HRESULT
VAR_INPUT
	hdl : UDINT; // Do not change, used by server.
END_VAR
callCounterAbort := callCounterAbort + 1;
END_METHOD

{attribute 'TcRpcEnable' := '1'}
METHOD CheckState : HRESULT
VAR_INPUT
	hdl : UDINT; // Do not change, used by server.
END_VAR
VAR_OUTPUT
	bBusy : BOOL; // Do not change. Used by server to find out if the job is finished
	
	// List of OutputArguments for OPC UA method, may be customized
	State : BOOL; // Abgeschlossener MethodCall
	MethodCall: BOOL; //Input Recall
END_VAR
callCounterCheckState := callCounterCheckState + 1;
IF NOT jobFinished THEN
	bBusy := TRUE; // job is not finished yet
	CheckState := 0; // no error
ELSE
	bBusy := FALSE; // job is finished
	CheckState := 0; // done, no error occured during execution (OPC UA StatusCode "GOOD")
	jobFinished := FALSE;
	State := ResetCall;
	MethodCall := MethodCall_HorizontalMove;
END_IF
END_METHOD

{attribute 'TcRpcEnable' := '1'}
METHOD Start : HRESULT
VAR_INPUT
	// List of InputArguments for OPC UA method, may be customized
	MethodCall : BOOL; // some description
	DirectionPoint : BOOL;
	EndschalterEntlastung : BOOL;	
END_VAR
VAR_OUTPUT
	hdl : UDINT; // Do not change, used by server.
END_VAR
callCounterStart := callCounterStart + 1;

MethodCall_HorizontalMove := MethodCall;
DirectionPoint := Direction;
EndschalterEntlastung := EndschalterEntlastung;

jobRunning := TRUE;
Start := 0; // no error occured, e.g. while parsing the input arguments (0 = OPC UA StatusCode "GOOD")
END_METHOD

END_FUNCTION_BLOCK

// ---- POUs/Moduls/MBS_Skills/MBS_DmPD_AS_RotationMove.TcPOU
{attribute 'OPC.UA.DA.JobMethod' := 'JobMethode_RotationMove'}
FUNCTION_BLOCK MBS_DmPD_AS_RotationMove
VAR
	AlwaysTrue : BOOL := TRUE;
	// Used for debugging purposes to display InputArguments of method call
	MethodCall_RotationMove : BOOL := FALSE; // used to store InputArg "MethodCall" from Start() method
	Direction : BOOL := FALSE;
	//	TS_EndschalterEntlastung : BOOL;
	callCounterStart : ULINT; // counts how many times the Start() method has been called
	callCounterCheckState : ULINT; // counts how many times the CheckState() method has been called
	callCounterAbort : ULINT; // counts how many times the Abort() method has been called
	
	// Variables to determine if a job has been started (Start() method has been called) or finished
	jobRunning : BOOL;
	jobFinished : BOOL;

	// State machine variable
	state : UDINT;
	
	//Variablen des Transport FBs
	ResetCall : BOOL := FALSE;	
	MBS_PD_RotationMove : AxisControl_MultipleInputSensors;
END_VAR
	
VAR_INPUT
	NotAusSignal: BOOL;
	LightSensor_01 : BOOL;
	LightSensor_02 : BOOL;
	TS_Endschalter_01 : BOOL;
	TS_Endschalter_02 : BOOL;
	TOF_Time_Motoransteuerung : TIME;
	TOF_Time_EndschalterEntlastung : TIME;
END_VAR

VAR_OUTPUT
	Motor_Ansteuerung01 : BOOL;
	Motor_Ansteuerung02 : BOOL;
END_VAR

